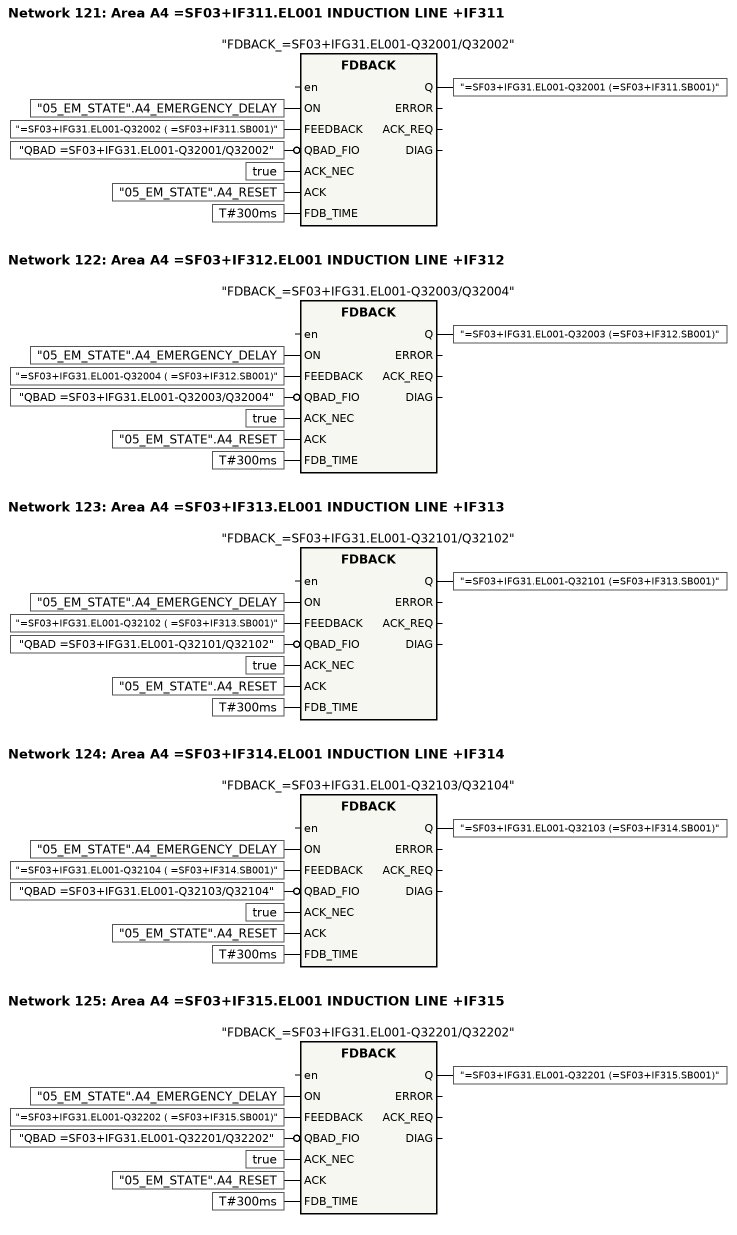
   "FDBACK_=SF03+IFG31.EL001-Q32001/Q32002"(ON := "05_EM_STATE".A4_EMERGENCY_DELAY,   // FDBACK
                           FEEDBACK := "=SF03+IFG31.EL001-Q32002 ( =SF03+IF311.SB001)",
                           QBAD_FIO := NOT "QBAD =SF03+IFG31.EL001-Q32001/Q32002",
                           ACK_NEC := true,
                           ACK := "05_EM_STATE".A4_RESET,
                           FDB_TIME := T#300ms,
                           Q => "=SF03+IFG31.EL001-Q32001 (=SF03+IF311.SB001)");
END_REGION

REGION Network 122: Area A4 =SF03+IF312.EL001 INDUCTION LINE +IF312
   "FDBACK_=SF03+IFG31.EL001-Q32003/Q32004"(ON := "05_EM_STATE".A4_EMERGENCY_DELAY,   // FDBACK
                           FEEDBACK := "=SF03+IFG31.EL001-Q32004 ( =SF03+IF312.SB001)",
                           QBAD_FIO := NOT "QBAD =SF03+IFG31.EL001-Q32003/Q32004",
                           ACK_NEC := true,
                           ACK := "05_EM_STATE".A4_RESET,
                           FDB_TIME := T#300ms,
                           Q => "=SF03+IFG31.EL001-Q32003 (=SF03+IF312.SB001)");
END_REGION

REGION Network 123: Area A4 =SF03+IF313.EL001 INDUCTION LINE +IF313
   "FDBACK_=SF03+IFG31.EL001-Q32101/Q32102"(ON := "05_EM_STATE".A4_EMERGENCY_DELAY,   // FDBACK
                           FEEDBACK := "=SF03+IFG31.EL001-Q32102 ( =SF03+IF313.SB001)",
                           QBAD_FIO := NOT "QBAD =SF03+IFG31.EL001-Q32101/Q32102",
                           ACK_NEC := true,
                           ACK := "05_EM_STATE".A4_RESET,
                           FDB_TIME := T#300ms,
                           Q => "=SF03+IFG31.EL001-Q32101 (=SF03+IF313.SB001)");
END_REGION

REGION Network 124: Area A4 =SF03+IF314.EL001 INDUCTION LINE +IF314
   "FDBACK_=SF03+IFG31.EL001-Q32103/Q32104"(ON := "05_EM_STATE".A4_EMERGENCY_DELAY,   // FDBACK
                           FEEDBACK := "=SF03+IFG31.EL001-Q32104 ( =SF03+IF314.SB001)",
                           QBAD_FIO := NOT "QBAD =SF03+IFG31.EL001-Q32103/Q32104",
                           ACK_NEC := true,
                           ACK := "05_EM_STATE".A4_RESET,
                           FDB_TIME := T#300ms,
                           Q => "=SF03+IFG31.EL001-Q32103 (=SF03+IF314.SB001)");
END_REGION

REGION Network 125: Area A4 =SF03+IF315.EL001 INDUCTION LINE +IF315
   "FDBACK_=SF03+IFG31.EL001-Q32201/Q32202"(ON := "05_EM_STATE".A4_EMERGENCY_DELAY,   // FDBACK
                           FEEDBACK := "=SF03+IFG31.EL001-Q32202 ( =SF03+IF315.SB001)",
                           QBAD_FIO := NOT "QBAD =SF03+IFG31.EL001-Q32201/Q32202",
                           ACK_NEC := true,
                           ACK := "05_EM_STATE".A4_RESET,
                           FDB_TIME := T#300ms,
                           Q => "=SF03+IFG31.EL001-Q32201 (=SF03+IF315.SB001)");
END_REGION

REGION Network 126: Area A4 =SF04+IF411.EL001 INDUCTION LINE +IF411
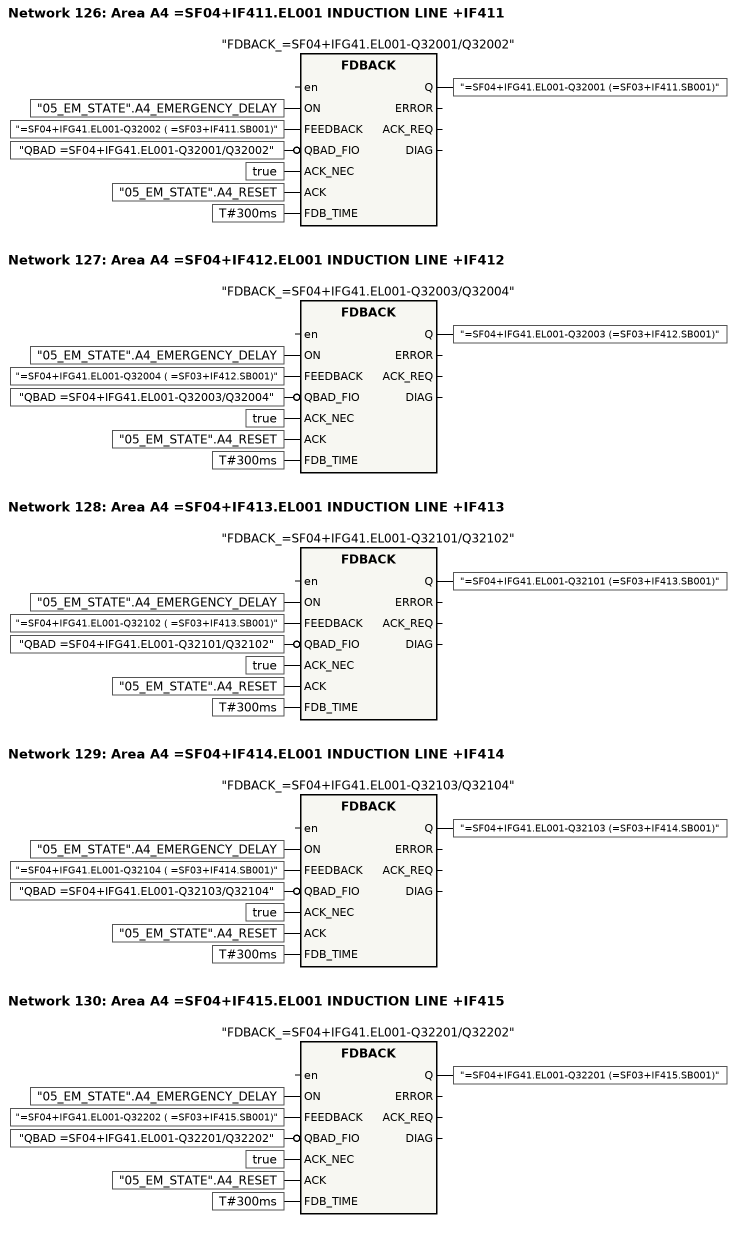
   "FDBACK_=SF04+IFG41.EL001-Q32001/Q32002"(ON := "05_EM_STATE".A4_EMERGENCY_DELAY,   // FDBACK
                           FEEDBACK := "=SF04+IFG41.EL001-Q32002 ( =SF03+IF411.SB001)",
                           QBAD_FIO := NOT "QBAD =SF04+IFG41.EL001-Q32001/Q32002",
                           ACK_NEC := true,
                           ACK := "05_EM_STATE".A4_RESET,
                           FDB_TIME := T#300ms,
                           Q => "=SF04+IFG41.EL001-Q32001 (=SF03+IF411.SB001)");
END_REGION

REGION Network 127: Area A4 =SF04+IF412.EL001 INDUCTION LINE +IF412
   "FDBACK_=SF04+IFG41.EL001-Q32003/Q32004"(ON := "05_EM_STATE".A4_EMERGENCY_DELAY,   // FDBACK
                           FEEDBACK := "=SF04+IFG41.EL001-Q32004 ( =SF03+IF412.SB001)",
                           QBAD_FIO := NOT "QBAD =SF04+IFG41.EL001-Q32003/Q32004",
                           ACK_NEC := true,
                           ACK := "05_EM_STATE".A4_RESET,
                           FDB_TIME := T#300ms,
                           Q => "=SF04+IFG41.EL001-Q32003 (=SF03+IF412.SB001)");
END_REGION

REGION Network 128: Area A4 =SF04+IF413.EL001 INDUCTION LINE +IF413
   "FDBACK_=SF04+IFG41.EL001-Q32101/Q32102"(ON := "05_EM_STATE".A4_EMERGENCY_DELAY,   // FDBACK
                           FEEDBACK := "=SF04+IFG41.EL001-Q32102 ( =SF03+IF413.SB001)",
                           QBAD_FIO := NOT "QBAD =SF04+IFG41.EL001-Q32101/Q32102",
                           ACK_NEC := true,
                           ACK := "05_EM_STATE".A4_RESET,
                           FDB_TIME := T#300ms,
                           Q => "=SF04+IFG41.EL001-Q32101 (=SF03+IF413.SB001)");
END_REGION

REGION Network 129: Area A4 =SF04+IF414.EL001 INDUCTION LINE +IF414
   "FDBACK_=SF04+IFG41.EL001-Q32103/Q32104"(ON := "05_EM_STATE".A4_EMERGENCY_DELAY,   // FDBACK
                           FEEDBACK := "=SF04+IFG41.EL001-Q32104 ( =SF03+IF414.SB001)",
                           QBAD_FIO := NOT "QBAD =SF04+IFG41.EL001-Q32103/Q32104",
                           ACK_NEC := true,
                           ACK := "05_EM_STATE".A4_RESET,
                           FDB_TIME := T#300ms,
                           Q => "=SF04+IFG41.EL001-Q32103 (=SF03+IF414.SB001)");
END_REGION

REGION Network 130: Area A4 =SF04+IF415.EL001 INDUCTION LINE +IF415
   "FDBACK_=SF04+IFG41.EL001-Q32201/Q32202"(ON := "05_EM_STATE".A4_EMERGENCY_DELAY,   // FDBACK
                           FEEDBACK := "=SF04+IFG41.EL001-Q32202 ( =SF03+IF415.SB001)",
                           QBAD_FIO := NOT "QBAD =SF04+IFG41.EL001-Q32201/Q32202",
                           ACK_NEC := true,
                           ACK := "05_EM_STATE".A4_RESET,
                           FDB_TIME := T#300ms,
                           Q => "=SF04+IFG41.EL001-Q32201 (=SF03+IF415.SB001)");
END_REGION

REGION Network 131: Area A4 =SF00+FC011.SB001 ROLLER CONVEYOR CHUTES +FH901/FH902
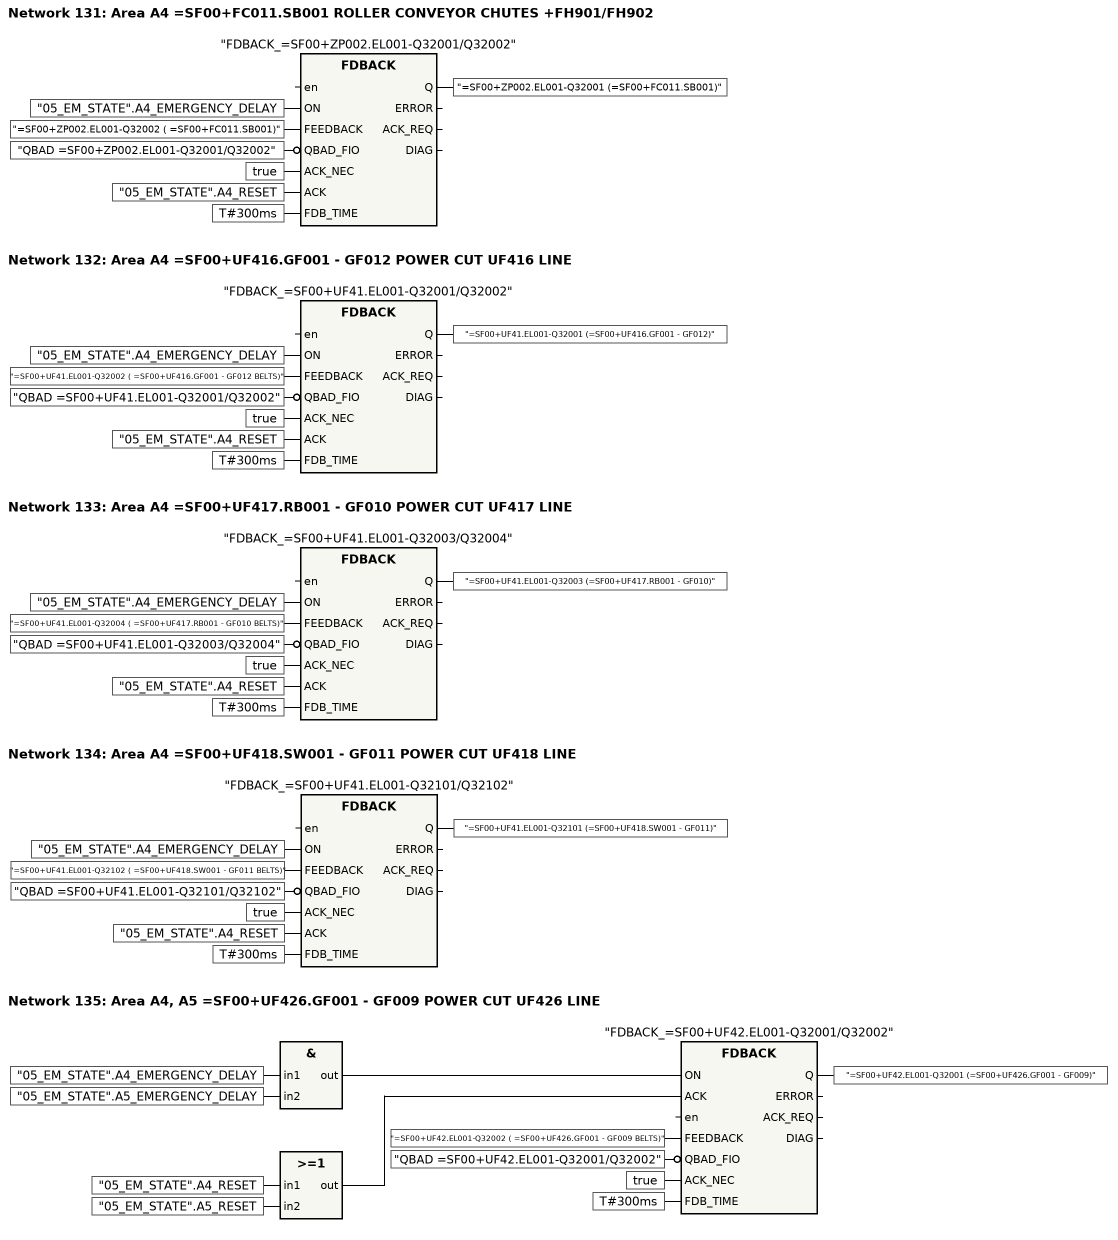
   "FDBACK_=SF00+ZP002.EL001-Q32001/Q32002"(ON := "05_EM_STATE".A4_EMERGENCY_DELAY,   // FDBACK
                           FEEDBACK := "=SF00+ZP002.EL001-Q32002 ( =SF00+FC011.SB001)",
                           QBAD_FIO := NOT "QBAD =SF00+ZP002.EL001-Q32001/Q32002",
                           ACK_NEC := true,
                           ACK := "05_EM_STATE".A4_RESET,
                           FDB_TIME := T#300ms,
                           Q => "=SF00+ZP002.EL001-Q32001 (=SF00+FC011.SB001)");
END_REGION

REGION Network 132: Area A4 =SF00+UF416.GF001 - GF012 POWER CUT UF416 LINE
   "FDBACK_=SF00+UF41.EL001-Q32001/Q32002"(ON := "05_EM_STATE".A4_EMERGENCY_DELAY,   // FDBACK
                           FEEDBACK := "=SF00+UF41.EL001-Q32002 ( =SF00+UF416.GF001 - GF012 BELTS)",
                           QBAD_FIO := NOT "QBAD =SF00+UF41.EL001-Q32001/Q32002",
                           ACK_NEC := true,
                           ACK := "05_EM_STATE".A4_RESET,
                           FDB_TIME := T#300ms,
                           Q => "=SF00+UF41.EL001-Q32001 (=SF00+UF416.GF001 - GF012)");
END_REGION

REGION Network 133: Area A4 =SF00+UF417.RB001 - GF010 POWER CUT UF417 LINE
   "FDBACK_=SF00+UF41.EL001-Q32003/Q32004"(ON := "05_EM_STATE".A4_EMERGENCY_DELAY,   // FDBACK
                           FEEDBACK := "=SF00+UF41.EL001-Q32004 ( =SF00+UF417.RB001 - GF010 BELTS)",
                           QBAD_FIO := NOT "QBAD =SF00+UF41.EL001-Q32003/Q32004",
                           ACK_NEC := true,
                           ACK := "05_EM_STATE".A4_RESET,
                           FDB_TIME := T#300ms,
                           Q => "=SF00+UF41.EL001-Q32003 (=SF00+UF417.RB001 - GF010)");
END_REGION

REGION Network 134: Area A4 =SF00+UF418.SW001 - GF011 POWER CUT UF418 LINE
   "FDBACK_=SF00+UF41.EL001-Q32101/Q32102"(ON := "05_EM_STATE".A4_EMERGENCY_DELAY,   // FDBACK
                           FEEDBACK := "=SF00+UF41.EL001-Q32102 ( =SF00+UF418.SW001 - GF011 BELTS)",
                           QBAD_FIO := NOT "QBAD =SF00+UF41.EL001-Q32101/Q32102",
                           ACK_NEC := true,
                           ACK := "05_EM_STATE".A4_RESET,
                           FDB_TIME := T#300ms,
                           Q => "=SF00+UF41.EL001-Q32101 (=SF00+UF418.SW001 - GF011)");
END_REGION

REGION Network 135: Area A4, A5 =SF00+UF426.GF001 - GF009 POWER CUT UF426 LINE
   "FDBACK_=SF00+UF42.EL001-Q32001/Q32002"(ON := "05_EM_STATE".A4_EMERGENCY_DELAY AND "05_EM_STATE".A5_EMERGENCY_DELAY,   // FDBACK
                           ACK := "05_EM_STATE".A4_RESET OR "05_EM_STATE".A5_RESET,
                           FEEDBACK := "=SF00+UF42.EL001-Q32002 ( =SF00+UF426.GF001 - GF009 BELTS)",
                           QBAD_FIO := NOT "QBAD =SF00+UF42.EL001-Q32001/Q32002",
                           ACK_NEC := true,
                           FDB_TIME := T#300ms,
                           Q => "=SF00+UF42.EL001-Q32001 (=SF00+UF426.GF001 - GF009)");
END_REGION

REGION Network 136: Area A4 =SF00+UF428.RB001 - GF010 POWER CUT UF428 LINE
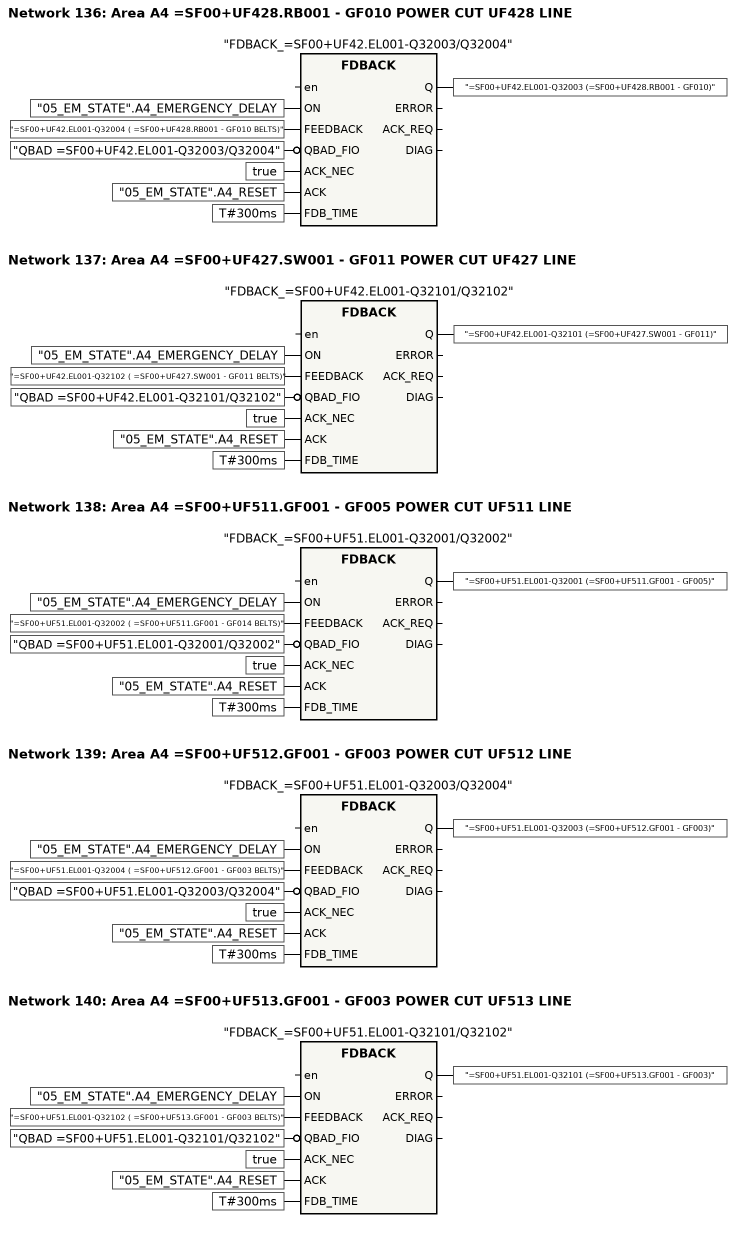
   "FDBACK_=SF00+UF42.EL001-Q32003/Q32004"(ON := "05_EM_STATE".A4_EMERGENCY_DELAY,   // FDBACK
                           FEEDBACK := "=SF00+UF42.EL001-Q32004 ( =SF00+UF428.RB001 - GF010 BELTS)",
                           QBAD_FIO := NOT "QBAD =SF00+UF42.EL001-Q32003/Q32004",
                           ACK_NEC := true,
                           ACK := "05_EM_STATE".A4_RESET,
                           FDB_TIME := T#300ms,
                           Q => "=SF00+UF42.EL001-Q32003 (=SF00+UF428.RB001 - GF010)");
END_REGION

REGION Network 137: Area A4 =SF00+UF427.SW001 - GF011 POWER CUT UF427 LINE
   "FDBACK_=SF00+UF42.EL001-Q32101/Q32102"(ON := "05_EM_STATE".A4_EMERGENCY_DELAY,   // FDBACK
                           FEEDBACK := "=SF00+UF42.EL001-Q32102 ( =SF00+UF427.SW001 - GF011 BELTS)",
                           QBAD_FIO := NOT "QBAD =SF00+UF42.EL001-Q32101/Q32102",
                           ACK_NEC := true,
                           ACK := "05_EM_STATE".A4_RESET,
                           FDB_TIME := T#300ms,
                           Q => "=SF00+UF42.EL001-Q32101 (=SF00+UF427.SW001 - GF011)");
END_REGION

REGION Network 138: Area A4 =SF00+UF511.GF001 - GF005 POWER CUT UF511 LINE
   "FDBACK_=SF00+UF51.EL001-Q32001/Q32002"(ON := "05_EM_STATE".A4_EMERGENCY_DELAY,   // FDBACK
                           FEEDBACK := "=SF00+UF51.EL001-Q32002 ( =SF00+UF511.GF001 - GF014 BELTS)",
                           QBAD_FIO := NOT "QBAD =SF00+UF51.EL001-Q32001/Q32002",
                           ACK_NEC := true,
                           ACK := "05_EM_STATE".A4_RESET,
                           FDB_TIME := T#300ms,
                           Q => "=SF00+UF51.EL001-Q32001 (=SF00+UF511.GF001 - GF005)");
END_REGION

REGION Network 139: Area A4 =SF00+UF512.GF001 - GF003 POWER CUT UF512 LINE
   "FDBACK_=SF00+UF51.EL001-Q32003/Q32004"(ON := "05_EM_STATE".A4_EMERGENCY_DELAY,   // FDBACK
                           FEEDBACK := "=SF00+UF51.EL001-Q32004 ( =SF00+UF512.GF001 - GF003 BELTS)",
                           QBAD_FIO := NOT "QBAD =SF00+UF51.EL001-Q32003/Q32004",
                           ACK_NEC := true,
                           ACK := "05_EM_STATE".A4_RESET,
                           FDB_TIME := T#300ms,
                           Q => "=SF00+UF51.EL001-Q32003 (=SF00+UF512.GF001 - GF003)");
END_REGION

REGION Network 140: Area A4 =SF00+UF513.GF001 - GF003 POWER CUT UF513 LINE
   "FDBACK_=SF00+UF51.EL001-Q32101/Q32102"(ON := "05_EM_STATE".A4_EMERGENCY_DELAY,   // FDBACK
                           FEEDBACK := "=SF00+UF51.EL001-Q32102 ( =SF00+UF513.GF001 - GF003 BELTS)",
                           QBAD_FIO := NOT "QBAD =SF00+UF51.EL001-Q32101/Q32102",
                           ACK_NEC := true,
                           ACK := "05_EM_STATE".A4_RESET,
                           FDB_TIME := T#300ms,
                           Q => "=SF00+UF51.EL001-Q32101 (=SF00+UF513.GF001 - GF003)");
END_REGION

REGION Network 141: Area A4, L15 =SF00+UF511.VS015 POWER CUT UF511 VERTICAL SWITCH
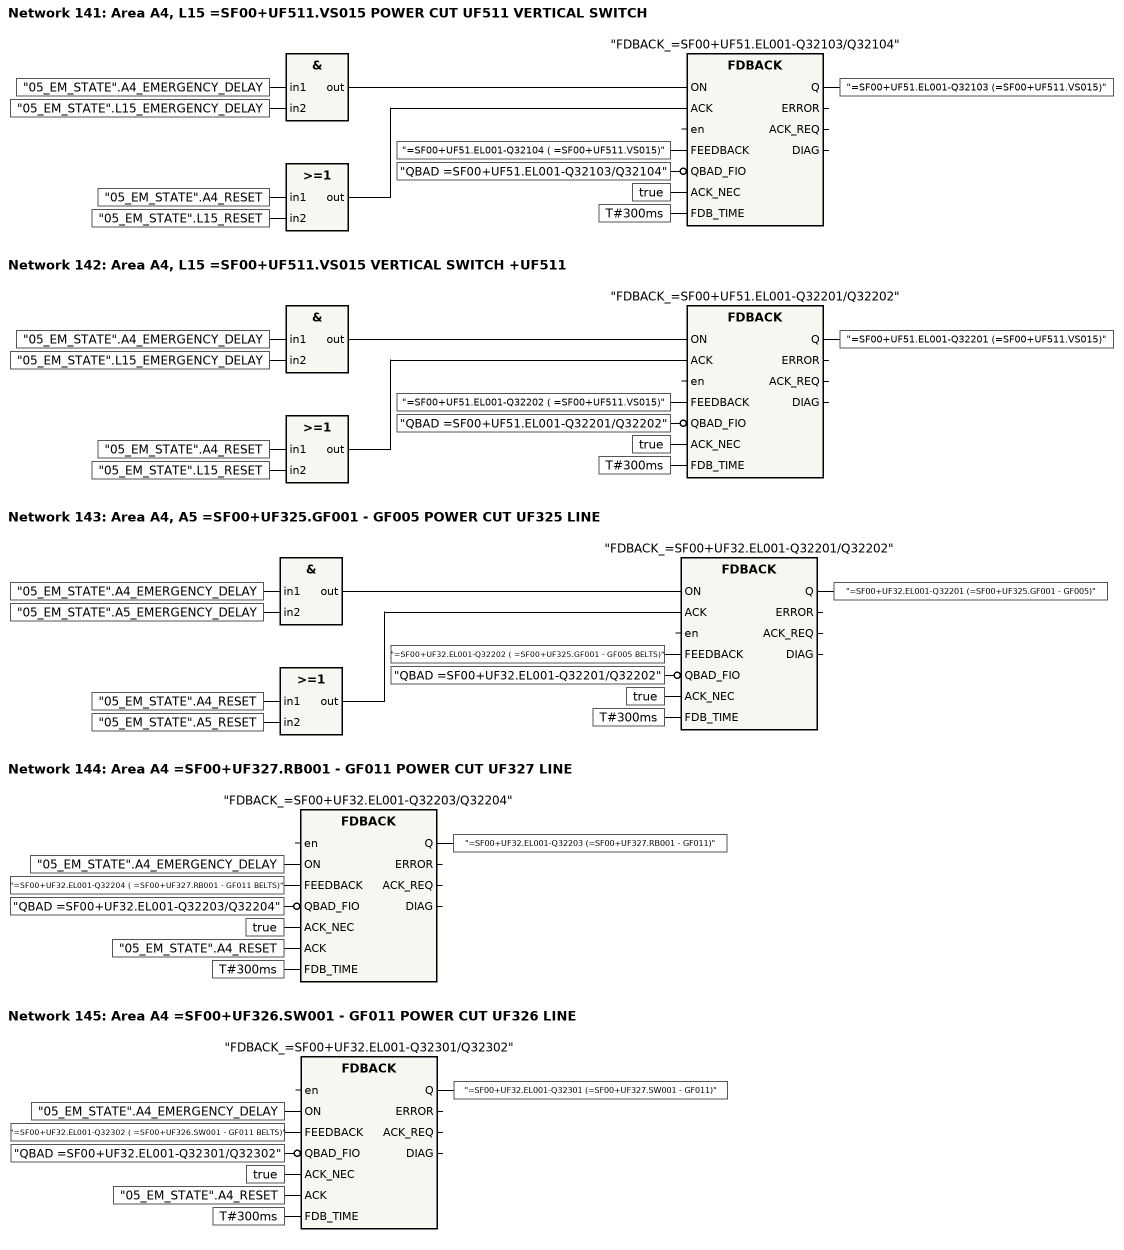
   "FDBACK_=SF00+UF51.EL001-Q32103/Q32104"(ON := "05_EM_STATE".A4_EMERGENCY_DELAY AND "05_EM_STATE".L15_EMERGENCY_DELAY,   // FDBACK
                           ACK := "05_EM_STATE".A4_RESET OR "05_EM_STATE".L15_RESET,
                           FEEDBACK := "=SF00+UF51.EL001-Q32104 ( =SF00+UF511.VS015)",
                           QBAD_FIO := NOT "QBAD =SF00+UF51.EL001-Q32103/Q32104",
                           ACK_NEC := true,
                           FDB_TIME := T#300ms,
                           Q => "=SF00+UF51.EL001-Q32103 (=SF00+UF511.VS015)");
END_REGION

REGION Network 142: Area A4, L15 =SF00+UF511.VS015 VERTICAL SWITCH +UF511
   "FDBACK_=SF00+UF51.EL001-Q32201/Q32202"(ON := "05_EM_STATE".A4_EMERGENCY_DELAY AND "05_EM_STATE".L15_EMERGENCY_DELAY,   // FDBACK
                           ACK := "05_EM_STATE".A4_RESET OR "05_EM_STATE".L15_RESET,
                           FEEDBACK := "=SF00+UF51.EL001-Q32202 ( =SF00+UF511.VS015)",
                           QBAD_FIO := NOT "QBAD =SF00+UF51.EL001-Q32201/Q32202",
                           ACK_NEC := true,
                           FDB_TIME := T#300ms,
                           Q => "=SF00+UF51.EL001-Q32201 (=SF00+UF511.VS015)");
END_REGION

REGION Network 143: Area A4, A5 =SF00+UF325.GF001 - GF005 POWER CUT UF325 LINE
   "FDBACK_=SF00+UF32.EL001-Q32201/Q32202"(ON := "05_EM_STATE".A4_EMERGENCY_DELAY AND "05_EM_STATE".A5_EMERGENCY_DELAY,   // FDBACK
                           ACK := "05_EM_STATE".A4_RESET OR "05_EM_STATE".A5_RESET,
                           FEEDBACK := "=SF00+UF32.EL001-Q32202 ( =SF00+UF325.GF001 - GF005 BELTS)",
                           QBAD_FIO := NOT "QBAD =SF00+UF32.EL001-Q32201/Q32202",
                           ACK_NEC := true,
                           FDB_TIME := T#300ms,
                           Q => "=SF00+UF32.EL001-Q32201 (=SF00+UF325.GF001 - GF005)");
END_REGION

REGION Network 144: Area A4 =SF00+UF327.RB001 - GF011 POWER CUT UF327 LINE
   "FDBACK_=SF00+UF32.EL001-Q32203/Q32204"(ON := "05_EM_STATE".A4_EMERGENCY_DELAY,   // FDBACK
                           FEEDBACK := "=SF00+UF32.EL001-Q32204 ( =SF00+UF327.RB001 - GF011 BELTS)",
                           QBAD_FIO := NOT "QBAD =SF00+UF32.EL001-Q32203/Q32204",
                           ACK_NEC := true,
                           ACK := "05_EM_STATE".A4_RESET,
                           FDB_TIME := T#300ms,
                           Q => "=SF00+UF32.EL001-Q32203 (=SF00+UF327.RB001 - GF011)");
END_REGION

REGION Network 145: Area A4 =SF00+UF326.SW001 - GF011 POWER CUT UF326 LINE
   "FDBACK_=SF00+UF32.EL001-Q32301/Q32302"(ON := "05_EM_STATE".A4_EMERGENCY_DELAY,   // FDBACK
                           FEEDBACK := "=SF00+UF32.EL001-Q32302 ( =SF00+UF326.SW001 - GF011 BELTS)",
                           QBAD_FIO := NOT "QBAD =SF00+UF32.EL001-Q32301/Q32302",
                           ACK_NEC := true,
                           ACK := "05_EM_STATE".A4_RESET,
                           FDB_TIME := T#300ms,
                           Q => "=SF00+UF32.EL001-Q32301 (=SF00+UF327.SW001 - GF011)");
END_REGION

REGION Network 146: Area A4 =SF00+UF317.GF001 - GF012 POWER CUT UF317 LINE
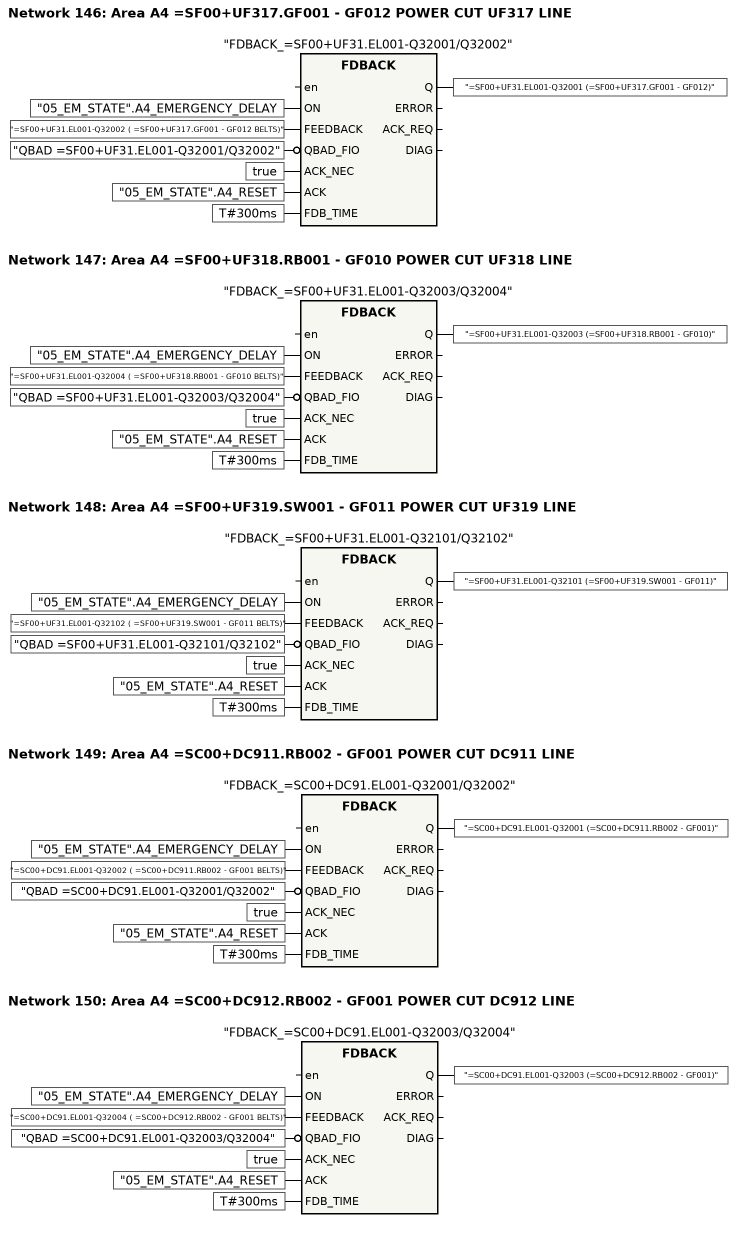
   "FDBACK_=SF00+UF31.EL001-Q32001/Q32002"(ON := "05_EM_STATE".A4_EMERGENCY_DELAY,   // FDBACK
                           FEEDBACK := "=SF00+UF31.EL001-Q32002 ( =SF00+UF317.GF001 - GF012 BELTS)",
                           QBAD_FIO := NOT "QBAD =SF00+UF31.EL001-Q32001/Q32002",
                           ACK_NEC := true,
                           ACK := "05_EM_STATE".A4_RESET,
                           FDB_TIME := T#300ms,
                           Q => "=SF00+UF31.EL001-Q32001 (=SF00+UF317.GF001 - GF012)");
END_REGION

REGION Network 147: Area A4 =SF00+UF318.RB001 - GF010 POWER CUT UF318 LINE
   "FDBACK_=SF00+UF31.EL001-Q32003/Q32004"(ON := "05_EM_STATE".A4_EMERGENCY_DELAY,   // FDBACK
                           FEEDBACK := "=SF00+UF31.EL001-Q32004 ( =SF00+UF318.RB001 - GF010 BELTS)",
                           QBAD_FIO := NOT "QBAD =SF00+UF31.EL001-Q32003/Q32004",
                           ACK_NEC := true,
                           ACK := "05_EM_STATE".A4_RESET,
                           FDB_TIME := T#300ms,
                           Q => "=SF00+UF31.EL001-Q32003 (=SF00+UF318.RB001 - GF010)");
END_REGION

REGION Network 148: Area A4 =SF00+UF319.SW001 - GF011 POWER CUT UF319 LINE
   "FDBACK_=SF00+UF31.EL001-Q32101/Q32102"(ON := "05_EM_STATE".A4_EMERGENCY_DELAY,   // FDBACK
                           FEEDBACK := "=SF00+UF31.EL001-Q32102 ( =SF00+UF319.SW001 - GF011 BELTS)",
                           QBAD_FIO := NOT "QBAD =SF00+UF31.EL001-Q32101/Q32102",
                           ACK_NEC := true,
                           ACK := "05_EM_STATE".A4_RESET,
                           FDB_TIME := T#300ms,
                           Q => "=SF00+UF31.EL001-Q32101 (=SF00+UF319.SW001 - GF011)");
END_REGION

REGION Network 149: Area A4 =SC00+DC911.RB002 - GF001 POWER CUT DC911 LINE
   "FDBACK_=SC00+DC91.EL001-Q32001/Q32002"(ON := "05_EM_STATE".A4_EMERGENCY_DELAY,   // FDBACK
                           FEEDBACK := "=SC00+DC91.EL001-Q32002 ( =SC00+DC911.RB002 - GF001 BELTS)",
                           QBAD_FIO := NOT "QBAD =SC00+DC91.EL001-Q32001/Q32002",
                           ACK_NEC := true,
                           ACK := "05_EM_STATE".A4_RESET,
                           FDB_TIME := T#300ms,
                           Q => "=SC00+DC91.EL001-Q32001 (=SC00+DC911.RB002 - GF001)");
END_REGION

REGION Network 150: Area A4 =SC00+DC912.RB002 - GF001 POWER CUT DC912 LINE
   "FDBACK_=SC00+DC91.EL001-Q32003/Q32004"(ON := "05_EM_STATE".A4_EMERGENCY_DELAY,   // FDBACK
                           FEEDBACK := "=SC00+DC91.EL001-Q32004 ( =SC00+DC912.RB002 - GF001 BELTS)",
                           QBAD_FIO := NOT "QBAD =SC00+DC91.EL001-Q32003/Q32004",
                           ACK_NEC := true,
                           ACK := "05_EM_STATE".A4_RESET,
                           FDB_TIME := T#300ms,
                           Q => "=SC00+DC91.EL001-Q32003 (=SC00+DC912.RB002 - GF001)");
END_REGION

REGION Network 151: Area A4 =SC00+DC913.RB002 - GF001 POWER CUT DC913 LINE
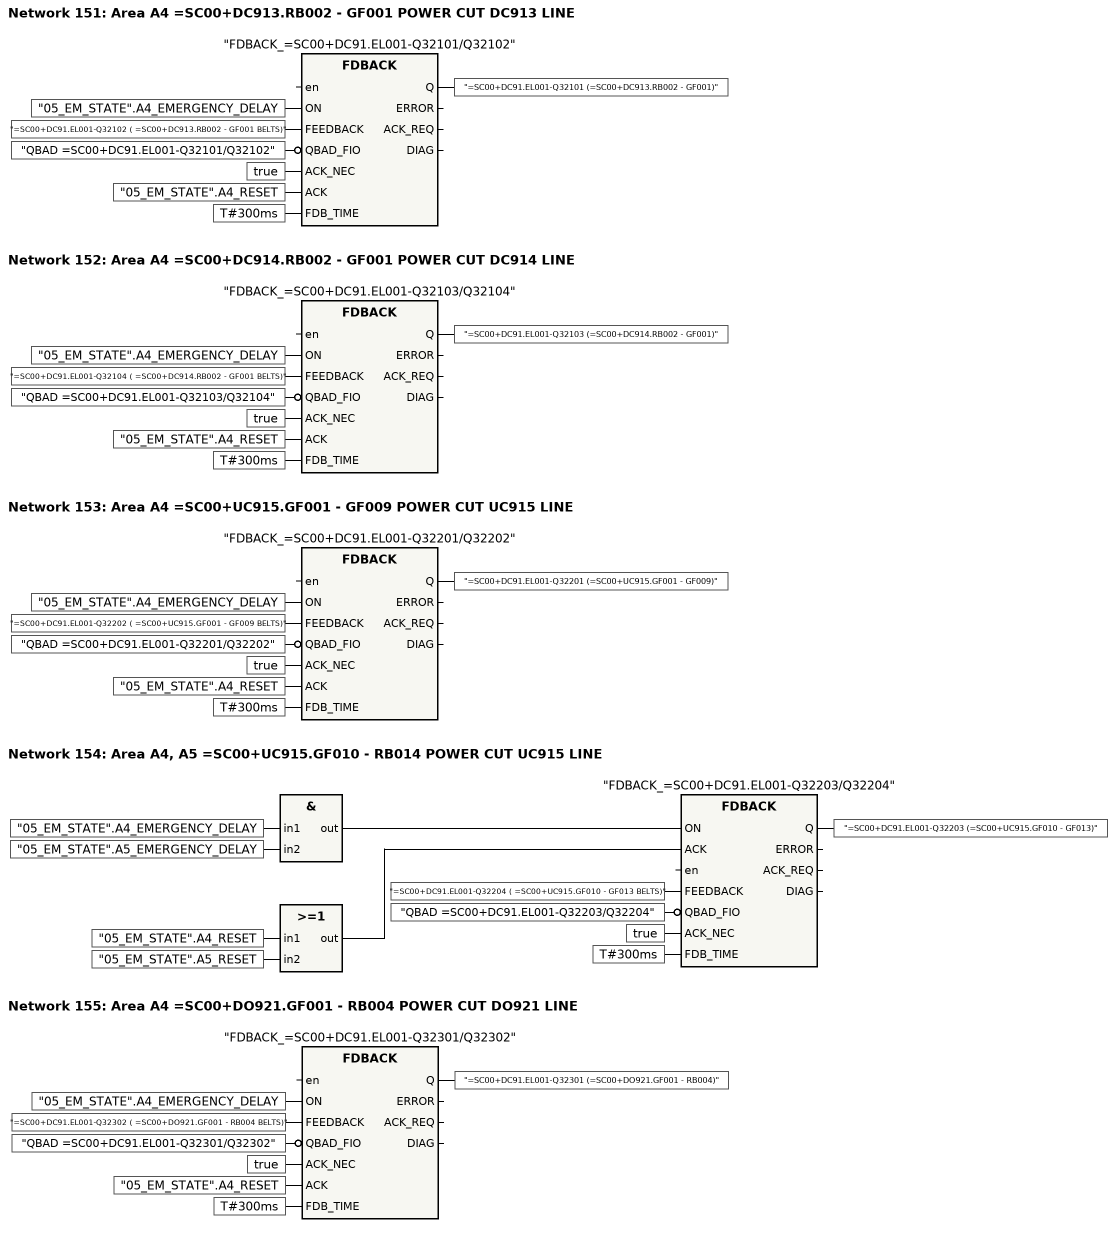
   "FDBACK_=SC00+DC91.EL001-Q32101/Q32102"(ON := "05_EM_STATE".A4_EMERGENCY_DELAY,   // FDBACK
                           FEEDBACK := "=SC00+DC91.EL001-Q32102 ( =SC00+DC913.RB002 - GF001 BELTS)",
                           QBAD_FIO := NOT "QBAD =SC00+DC91.EL001-Q32101/Q32102",
                           ACK_NEC := true,
                           ACK := "05_EM_STATE".A4_RESET,
                           FDB_TIME := T#300ms,
                           Q => "=SC00+DC91.EL001-Q32101 (=SC00+DC913.RB002 - GF001)");
END_REGION

REGION Network 152: Area A4 =SC00+DC914.RB002 - GF001 POWER CUT DC914 LINE
   "FDBACK_=SC00+DC91.EL001-Q32103/Q32104"(ON := "05_EM_STATE".A4_EMERGENCY_DELAY,   // FDBACK
                           FEEDBACK := "=SC00+DC91.EL001-Q32104 ( =SC00+DC914.RB002 - GF001 BELTS)",
                           QBAD_FIO := NOT "QBAD =SC00+DC91.EL001-Q32103/Q32104",
                           ACK_NEC := true,
                           ACK := "05_EM_STATE".A4_RESET,
                           FDB_TIME := T#300ms,
                           Q => "=SC00+DC91.EL001-Q32103 (=SC00+DC914.RB002 - GF001)");
END_REGION

REGION Network 153: Area A4 =SC00+UC915.GF001 - GF009 POWER CUT UC915 LINE
   "FDBACK_=SC00+DC91.EL001-Q32201/Q32202"(ON := "05_EM_STATE".A4_EMERGENCY_DELAY,   // FDBACK
                           FEEDBACK := "=SC00+DC91.EL001-Q32202 ( =SC00+UC915.GF001 - GF009 BELTS)",
                           QBAD_FIO := NOT "QBAD =SC00+DC91.EL001-Q32201/Q32202",
                           ACK_NEC := true,
                           ACK := "05_EM_STATE".A4_RESET,
                           FDB_TIME := T#300ms,
                           Q => "=SC00+DC91.EL001-Q32201 (=SC00+UC915.GF001 - GF009)");
END_REGION

REGION Network 154: Area A4, A5 =SC00+UC915.GF010 - RB014 POWER CUT UC915 LINE
   "FDBACK_=SC00+DC91.EL001-Q32203/Q32204"(ON := "05_EM_STATE".A4_EMERGENCY_DELAY AND "05_EM_STATE".A5_EMERGENCY_DELAY,   // FDBACK
                           ACK := "05_EM_STATE".A4_RESET OR "05_EM_STATE".A5_RESET,
                           FEEDBACK := "=SC00+DC91.EL001-Q32204 ( =SC00+UC915.GF010 - GF013 BELTS)",
                           QBAD_FIO := NOT "QBAD =SC00+DC91.EL001-Q32203/Q32204",
                           ACK_NEC := true,
                           FDB_TIME := T#300ms,
                           Q => "=SC00+DC91.EL001-Q32203 (=SC00+UC915.GF010 - GF013)");
END_REGION

REGION Network 155: Area A4 =SC00+DO921.GF001 - RB004 POWER CUT DO921 LINE
   "FDBACK_=SC00+DC91.EL001-Q32301/Q32302"(ON := "05_EM_STATE".A4_EMERGENCY_DELAY,   // FDBACK
                           FEEDBACK := "=SC00+DC91.EL001-Q32302 ( =SC00+DO921.GF001 - RB004 BELTS)",
                           QBAD_FIO := NOT "QBAD =SC00+DC91.EL001-Q32301/Q32302",
                           ACK_NEC := true,
                           ACK := "05_EM_STATE".A4_RESET,
                           FDB_TIME := T#300ms,
                           Q => "=SC00+DC91.EL001-Q32301 (=SC00+DO921.GF001 - RB004)");
END_REGION

REGION Network 156: Area A4, A5 =SC00+UC291.GF001 - RB010 POWER CUT UC291 LINE
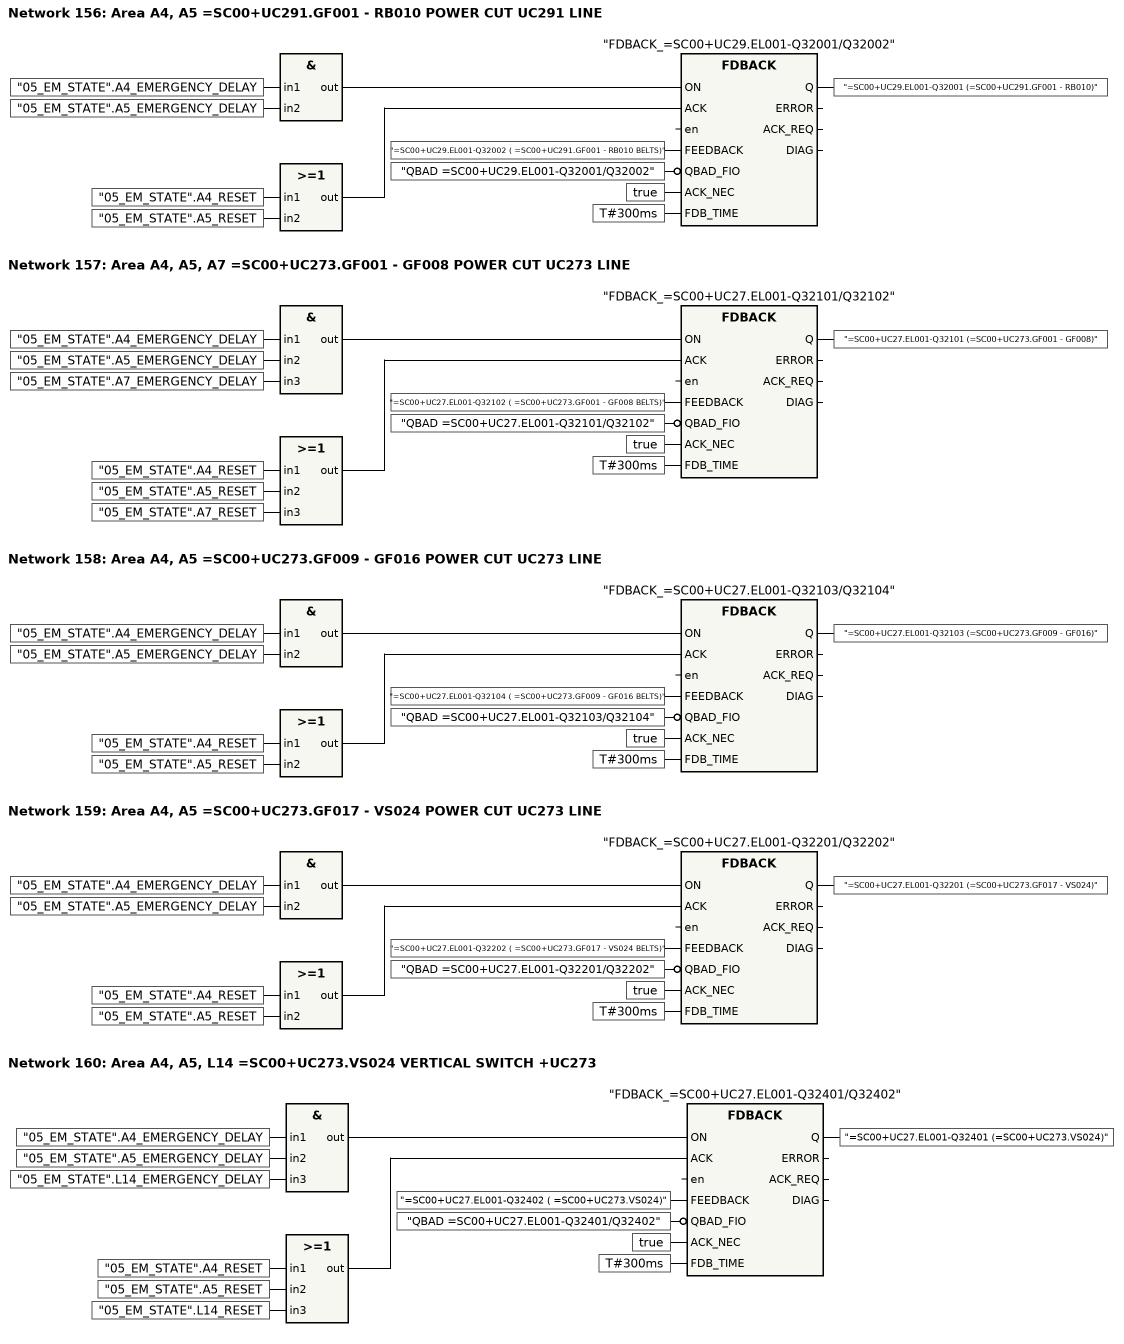
   "FDBACK_=SC00+UC29.EL001-Q32001/Q32002"(ON := "05_EM_STATE".A4_EMERGENCY_DELAY AND "05_EM_STATE".A5_EMERGENCY_DELAY,   // FDBACK
                           ACK := "05_EM_STATE".A4_RESET OR "05_EM_STATE".A5_RESET,
                           FEEDBACK := "=SC00+UC29.EL001-Q32002 ( =SC00+UC291.GF001 - RB010 BELTS)",
                           QBAD_FIO := NOT "QBAD =SC00+UC29.EL001-Q32001/Q32002",
                           ACK_NEC := true,
                           FDB_TIME := T#300ms,
                           Q => "=SC00+UC29.EL001-Q32001 (=SC00+UC291.GF001 - RB010)");
END_REGION

REGION Network 157: Area A4, A5, A7 =SC00+UC273.GF001 - GF008 POWER CUT UC273 LINE
   "FDBACK_=SC00+UC27.EL001-Q32101/Q32102"(ON := "05_EM_STATE".A4_EMERGENCY_DELAY AND "05_EM_STATE".A5_EMERGENCY_DELAY AND "05_EM_STATE".A7_EMERGENCY_DELAY,   // FDBACK
                           ACK := "05_EM_STATE".A4_RESET OR "05_EM_STATE".A5_RESET OR "05_EM_STATE".A7_RESET,
                           FEEDBACK := "=SC00+UC27.EL001-Q32102 ( =SC00+UC273.GF001 - GF008 BELTS)",
                           QBAD_FIO := NOT "QBAD =SC00+UC27.EL001-Q32101/Q32102",
                           ACK_NEC := true,
                           FDB_TIME := T#300ms,
                           Q => "=SC00+UC27.EL001-Q32101 (=SC00+UC273.GF001 - GF008)");
END_REGION

REGION Network 158: Area A4, A5 =SC00+UC273.GF009 - GF016 POWER CUT UC273 LINE
   "FDBACK_=SC00+UC27.EL001-Q32103/Q32104"(ON := "05_EM_STATE".A4_EMERGENCY_DELAY AND "05_EM_STATE".A5_EMERGENCY_DELAY,   // FDBACK
                           ACK := "05_EM_STATE".A4_RESET OR "05_EM_STATE".A5_RESET,
                           FEEDBACK := "=SC00+UC27.EL001-Q32104 ( =SC00+UC273.GF009 - GF016 BELTS)",
                           QBAD_FIO := NOT "QBAD =SC00+UC27.EL001-Q32103/Q32104",
                           ACK_NEC := true,
                           FDB_TIME := T#300ms,
                           Q => "=SC00+UC27.EL001-Q32103 (=SC00+UC273.GF009 - GF016)");
END_REGION

REGION Network 159: Area A4, A5 =SC00+UC273.GF017 - VS024 POWER CUT UC273 LINE
   "FDBACK_=SC00+UC27.EL001-Q32201/Q32202"(ON := "05_EM_STATE".A4_EMERGENCY_DELAY AND "05_EM_STATE".A5_EMERGENCY_DELAY,   // FDBACK
                           ACK := "05_EM_STATE".A4_RESET OR "05_EM_STATE".A5_RESET,
                           FEEDBACK := "=SC00+UC27.EL001-Q32202 ( =SC00+UC273.GF017 - VS024 BELTS)",
                           QBAD_FIO := NOT "QBAD =SC00+UC27.EL001-Q32201/Q32202",
                           ACK_NEC := true,
                           FDB_TIME := T#300ms,
                           Q => "=SC00+UC27.EL001-Q32201 (=SC00+UC273.GF017 - VS024)");
END_REGION

REGION Network 160: Area A4, A5, L14 =SC00+UC273.VS024 VERTICAL SWITCH +UC273
   "FDBACK_=SC00+UC27.EL001-Q32401/Q32402"(ON := "05_EM_STATE".A4_EMERGENCY_DELAY AND "05_EM_STATE".A5_EMERGENCY_DELAY AND "05_EM_STATE".L14_EMERGENCY_DELAY,   // FDBACK
                           ACK := "05_EM_STATE".A4_RESET OR "05_EM_STATE".A5_RESET OR "05_EM_STATE".L14_RESET,
                           FEEDBACK := "=SC00+UC27.EL001-Q32402 ( =SC00+UC273.VS024)",
                           QBAD_FIO := NOT "QBAD =SC00+UC27.EL001-Q32401/Q32402",
                           ACK_NEC := true,
                           FDB_TIME := T#300ms,
                           Q => "=SC00+UC27.EL001-Q32401 (=SC00+UC273.VS024)");
END_REGION

REGION Network 161: Area A4, A5, L14 =SC00+UC273.VS024 VERTICAL SWITCH +UC273
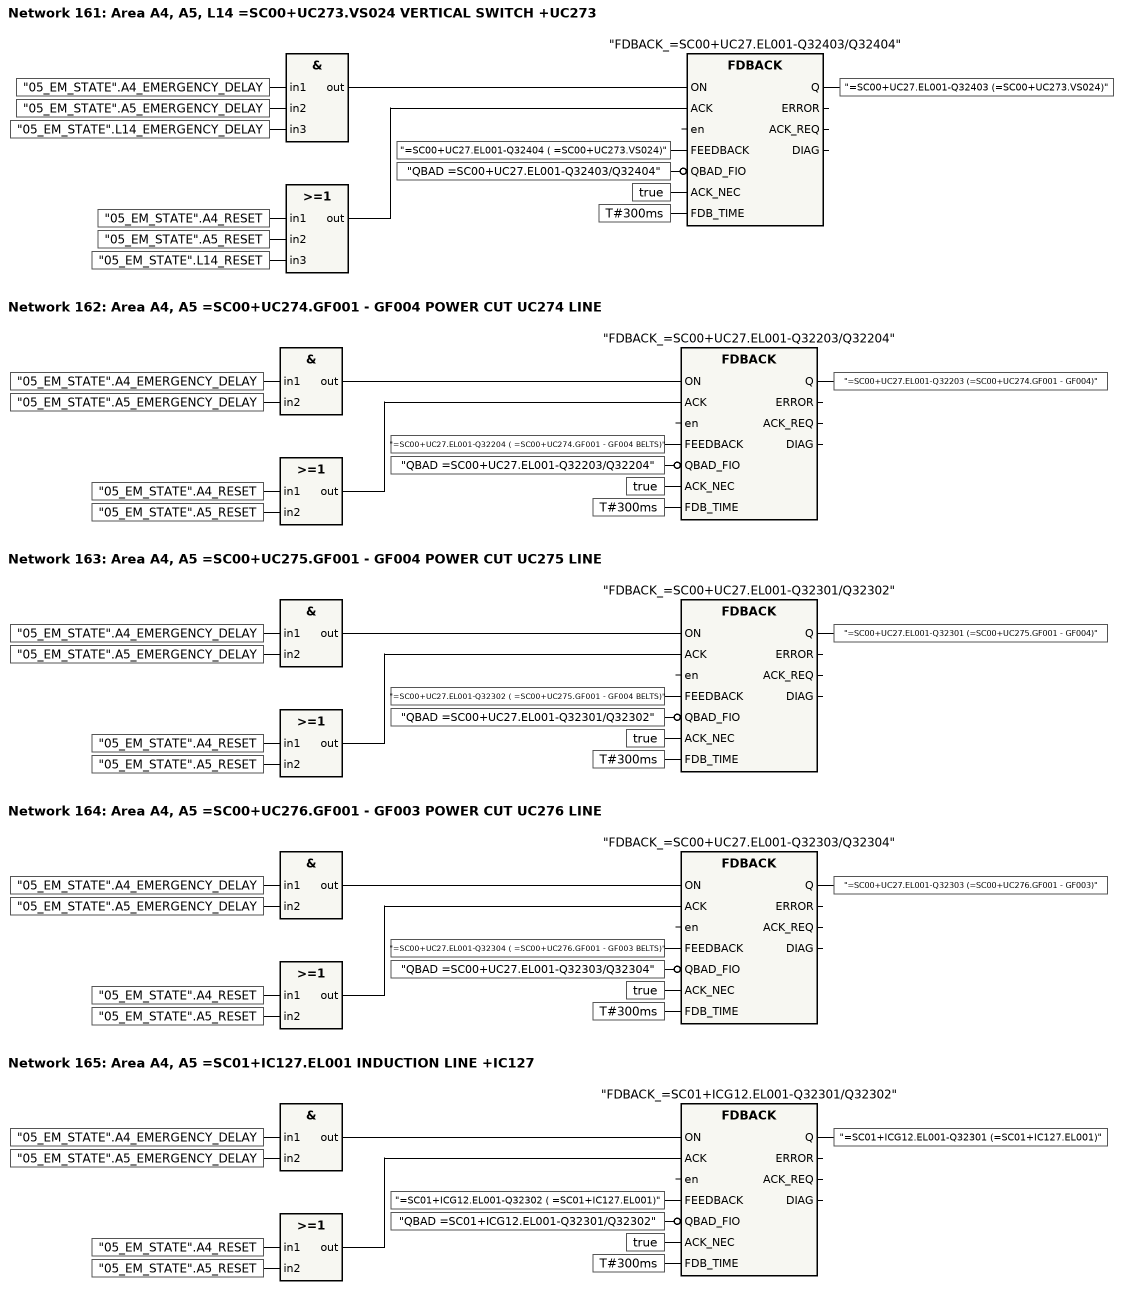
   "FDBACK_=SC00+UC27.EL001-Q32403/Q32404"(ON := "05_EM_STATE".A4_EMERGENCY_DELAY AND "05_EM_STATE".A5_EMERGENCY_DELAY AND "05_EM_STATE".L14_EMERGENCY_DELAY,   // FDBACK
                           ACK := "05_EM_STATE".A4_RESET OR "05_EM_STATE".A5_RESET OR "05_EM_STATE".L14_RESET,
                           FEEDBACK := "=SC00+UC27.EL001-Q32404 ( =SC00+UC273.VS024)",
                           QBAD_FIO := NOT "QBAD =SC00+UC27.EL001-Q32403/Q32404",
                           ACK_NEC := true,
                           FDB_TIME := T#300ms,
                           Q => "=SC00+UC27.EL001-Q32403 (=SC00+UC273.VS024)");
END_REGION

REGION Network 162: Area A4, A5 =SC00+UC274.GF001 - GF004 POWER CUT UC274 LINE
   "FDBACK_=SC00+UC27.EL001-Q32203/Q32204"(ON := "05_EM_STATE".A4_EMERGENCY_DELAY AND "05_EM_STATE".A5_EMERGENCY_DELAY,   // FDBACK
                           ACK := "05_EM_STATE".A4_RESET OR "05_EM_STATE".A5_RESET,
                           FEEDBACK := "=SC00+UC27.EL001-Q32204 ( =SC00+UC274.GF001 - GF004 BELTS)",
                           QBAD_FIO := NOT "QBAD =SC00+UC27.EL001-Q32203/Q32204",
                           ACK_NEC := true,
                           FDB_TIME := T#300ms,
                           Q => "=SC00+UC27.EL001-Q32203 (=SC00+UC274.GF001 - GF004)");
END_REGION

REGION Network 163: Area A4, A5 =SC00+UC275.GF001 - GF004 POWER CUT UC275 LINE
   "FDBACK_=SC00+UC27.EL001-Q32301/Q32302"(ON := "05_EM_STATE".A4_EMERGENCY_DELAY AND "05_EM_STATE".A5_EMERGENCY_DELAY,   // FDBACK
                           ACK := "05_EM_STATE".A4_RESET OR "05_EM_STATE".A5_RESET,
                           FEEDBACK := "=SC00+UC27.EL001-Q32302 ( =SC00+UC275.GF001 - GF004 BELTS)",
                           QBAD_FIO := NOT "QBAD =SC00+UC27.EL001-Q32301/Q32302",
                           ACK_NEC := true,
                           FDB_TIME := T#300ms,
                           Q => "=SC00+UC27.EL001-Q32301 (=SC00+UC275.GF001 - GF004)");
END_REGION

REGION Network 164: Area A4, A5 =SC00+UC276.GF001 - GF003 POWER CUT UC276 LINE
   "FDBACK_=SC00+UC27.EL001-Q32303/Q32304"(ON := "05_EM_STATE".A4_EMERGENCY_DELAY AND "05_EM_STATE".A5_EMERGENCY_DELAY,   // FDBACK
                           ACK := "05_EM_STATE".A4_RESET OR "05_EM_STATE".A5_RESET,
                           FEEDBACK := "=SC00+UC27.EL001-Q32304 ( =SC00+UC276.GF001 - GF003 BELTS)",
                           QBAD_FIO := NOT "QBAD =SC00+UC27.EL001-Q32303/Q32304",
                           ACK_NEC := true,
                           FDB_TIME := T#300ms,
                           Q => "=SC00+UC27.EL001-Q32303 (=SC00+UC276.GF001 - GF003)");
END_REGION

REGION Network 165: Area A4, A5 =SC01+IC127.EL001 INDUCTION LINE +IC127
   "FDBACK_=SC01+ICG12.EL001-Q32301/Q32302"(ON := "05_EM_STATE".A4_EMERGENCY_DELAY AND "05_EM_STATE".A5_EMERGENCY_DELAY,   // FDBACK
                           ACK := "05_EM_STATE".A4_RESET OR "05_EM_STATE".A5_RESET,
                           FEEDBACK := "=SC01+ICG12.EL001-Q32302 ( =SC01+IC127.EL001)",
                           QBAD_FIO := NOT "QBAD =SC01+ICG12.EL001-Q32301/Q32302",
                           ACK_NEC := true,
                           FDB_TIME := T#300ms,
                           Q => "=SC01+ICG12.EL001-Q32301 (=SC01+IC127.EL001)");
END_REGION

REGION Network 166: Area A4, A5 =SC02+IC227.EL001 INDUCTION LINE +IC227
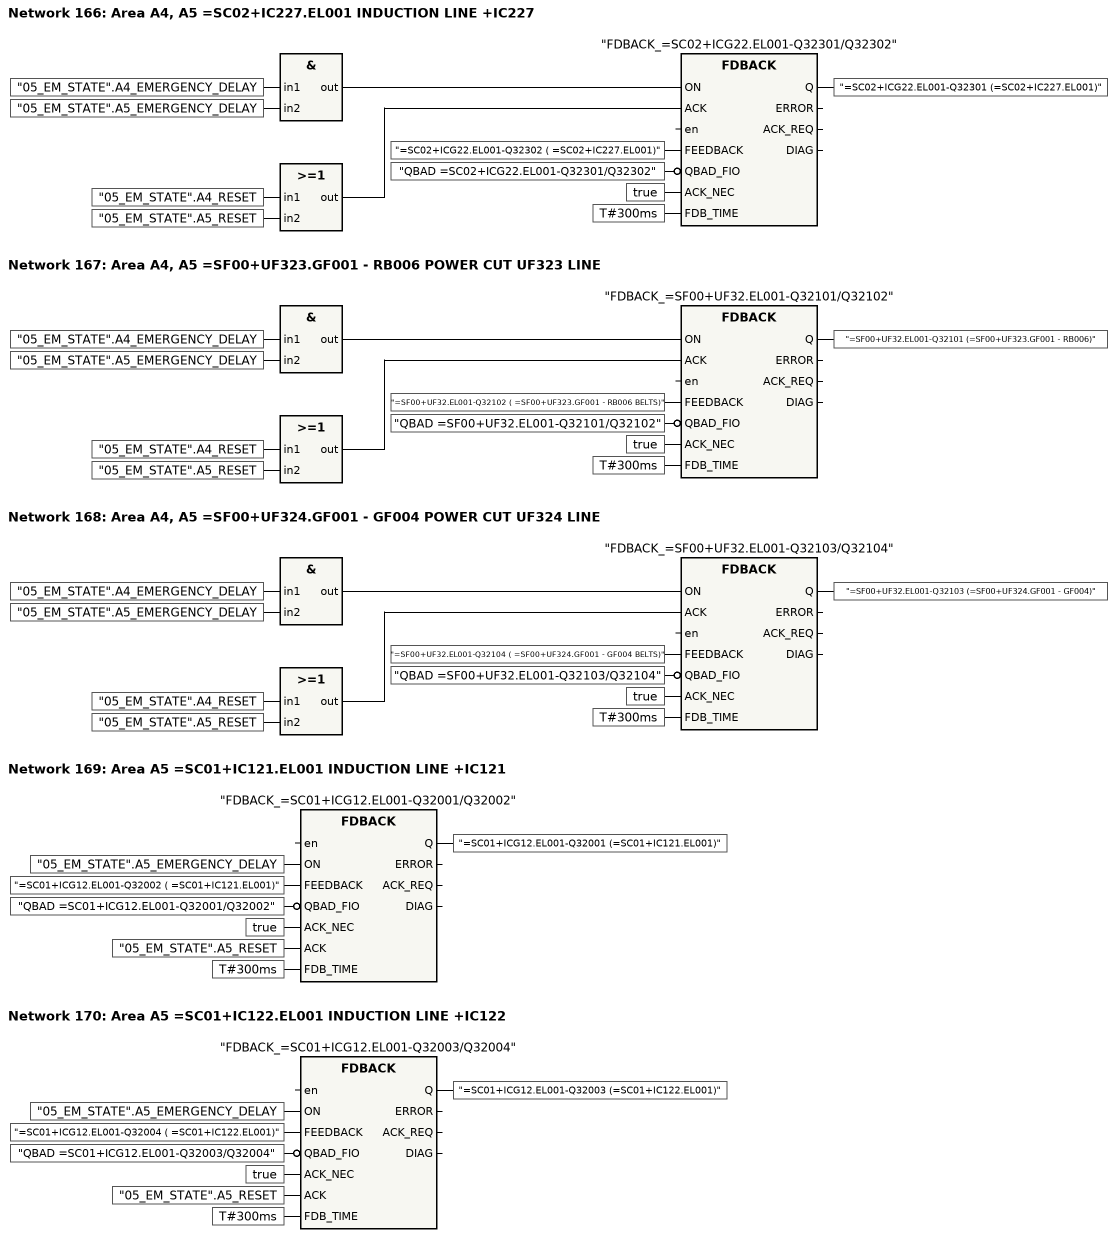
   "FDBACK_=SC02+ICG22.EL001-Q32301/Q32302"(ON := "05_EM_STATE".A4_EMERGENCY_DELAY AND "05_EM_STATE".A5_EMERGENCY_DELAY,   // FDBACK
                           ACK := "05_EM_STATE".A4_RESET OR "05_EM_STATE".A5_RESET,
                           FEEDBACK := "=SC02+ICG22.EL001-Q32302 ( =SC02+IC227.EL001)",
                           QBAD_FIO := NOT "QBAD =SC02+ICG22.EL001-Q32301/Q32302",
                           ACK_NEC := true,
                           FDB_TIME := T#300ms,
                           Q => "=SC02+ICG22.EL001-Q32301 (=SC02+IC227.EL001)");
END_REGION

REGION Network 167: Area A4, A5 =SF00+UF323.GF001 - RB006 POWER CUT UF323 LINE
   "FDBACK_=SF00+UF32.EL001-Q32101/Q32102"(ON := "05_EM_STATE".A4_EMERGENCY_DELAY AND "05_EM_STATE".A5_EMERGENCY_DELAY,   // FDBACK
                           ACK := "05_EM_STATE".A4_RESET OR "05_EM_STATE".A5_RESET,
                           FEEDBACK := "=SF00+UF32.EL001-Q32102 ( =SF00+UF323.GF001 - RB006 BELTS)",
                           QBAD_FIO := NOT "QBAD =SF00+UF32.EL001-Q32101/Q32102",
                           ACK_NEC := true,
                           FDB_TIME := T#300ms,
                           Q => "=SF00+UF32.EL001-Q32101 (=SF00+UF323.GF001 - RB006)");
END_REGION

REGION Network 168: Area A4, A5 =SF00+UF324.GF001 - GF004 POWER CUT UF324 LINE
   "FDBACK_=SF00+UF32.EL001-Q32103/Q32104"(ON := "05_EM_STATE".A4_EMERGENCY_DELAY AND "05_EM_STATE".A5_EMERGENCY_DELAY,   // FDBACK
                           ACK := "05_EM_STATE".A4_RESET OR "05_EM_STATE".A5_RESET,
                           FEEDBACK := "=SF00+UF32.EL001-Q32104 ( =SF00+UF324.GF001 - GF004 BELTS)",
                           QBAD_FIO := NOT "QBAD =SF00+UF32.EL001-Q32103/Q32104",
                           ACK_NEC := true,
                           FDB_TIME := T#300ms,
                           Q => "=SF00+UF32.EL001-Q32103 (=SF00+UF324.GF001 - GF004)");
END_REGION

REGION Network 169: Area A5 =SC01+IC121.EL001 INDUCTION LINE +IC121
   "FDBACK_=SC01+ICG12.EL001-Q32001/Q32002"(ON := "05_EM_STATE".A5_EMERGENCY_DELAY,   // FDBACK
                           FEEDBACK := "=SC01+ICG12.EL001-Q32002 ( =SC01+IC121.EL001)",
                           QBAD_FIO := NOT "QBAD =SC01+ICG12.EL001-Q32001/Q32002",
                           ACK_NEC := true,
                           ACK := "05_EM_STATE".A5_RESET,
                           FDB_TIME := T#300ms,
                           Q => "=SC01+ICG12.EL001-Q32001 (=SC01+IC121.EL001)");
END_REGION

REGION Network 170: Area A5 =SC01+IC122.EL001 INDUCTION LINE +IC122
   "FDBACK_=SC01+ICG12.EL001-Q32003/Q32004"(ON := "05_EM_STATE".A5_EMERGENCY_DELAY,   // FDBACK
                           FEEDBACK := "=SC01+ICG12.EL001-Q32004 ( =SC01+IC122.EL001)",
                           QBAD_FIO := NOT "QBAD =SC01+ICG12.EL001-Q32003/Q32004",
                           ACK_NEC := true,
                           ACK := "05_EM_STATE".A5_RESET,
                           FDB_TIME := T#300ms,
                           Q => "=SC01+ICG12.EL001-Q32003 (=SC01+IC122.EL001)");
END_REGION

REGION Network 171: Area A5 =SC01+IC123.EL001 INDUCTION LINE +IC123
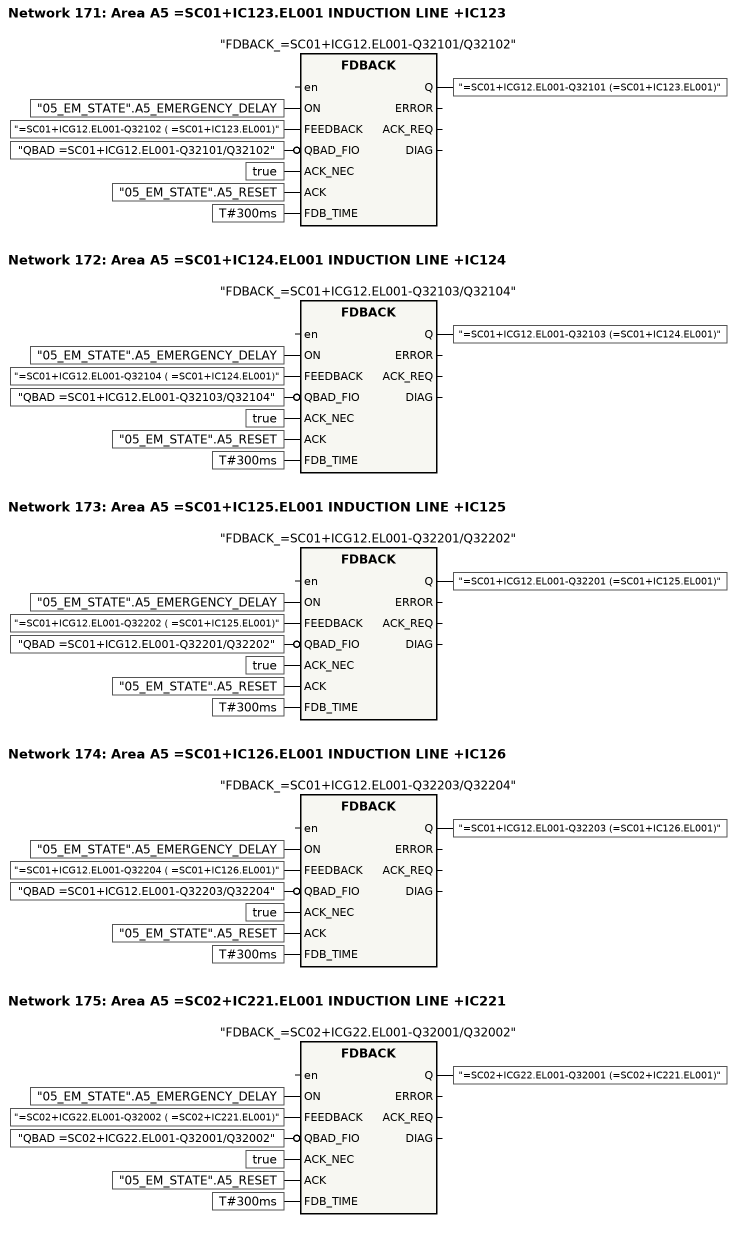
   "FDBACK_=SC01+ICG12.EL001-Q32101/Q32102"(ON := "05_EM_STATE".A5_EMERGENCY_DELAY,   // FDBACK
                           FEEDBACK := "=SC01+ICG12.EL001-Q32102 ( =SC01+IC123.EL001)",
                           QBAD_FIO := NOT "QBAD =SC01+ICG12.EL001-Q32101/Q32102",
                           ACK_NEC := true,
                           ACK := "05_EM_STATE".A5_RESET,
                           FDB_TIME := T#300ms,
                           Q => "=SC01+ICG12.EL001-Q32101 (=SC01+IC123.EL001)");
END_REGION

REGION Network 172: Area A5 =SC01+IC124.EL001 INDUCTION LINE +IC124
   "FDBACK_=SC01+ICG12.EL001-Q32103/Q32104"(ON := "05_EM_STATE".A5_EMERGENCY_DELAY,   // FDBACK
                           FEEDBACK := "=SC01+ICG12.EL001-Q32104 ( =SC01+IC124.EL001)",
                           QBAD_FIO := NOT "QBAD =SC01+ICG12.EL001-Q32103/Q32104",
                           ACK_NEC := true,
                           ACK := "05_EM_STATE".A5_RESET,
                           FDB_TIME := T#300ms,
                           Q => "=SC01+ICG12.EL001-Q32103 (=SC01+IC124.EL001)");
END_REGION

REGION Network 173: Area A5 =SC01+IC125.EL001 INDUCTION LINE +IC125
   "FDBACK_=SC01+ICG12.EL001-Q32201/Q32202"(ON := "05_EM_STATE".A5_EMERGENCY_DELAY,   // FDBACK
                           FEEDBACK := "=SC01+ICG12.EL001-Q32202 ( =SC01+IC125.EL001)",
                           QBAD_FIO := NOT "QBAD =SC01+ICG12.EL001-Q32201/Q32202",
                           ACK_NEC := true,
                           ACK := "05_EM_STATE".A5_RESET,
                           FDB_TIME := T#300ms,
                           Q => "=SC01+ICG12.EL001-Q32201 (=SC01+IC125.EL001)");
END_REGION

REGION Network 174: Area A5 =SC01+IC126.EL001 INDUCTION LINE +IC126
   "FDBACK_=SC01+ICG12.EL001-Q32203/Q32204"(ON := "05_EM_STATE".A5_EMERGENCY_DELAY,   // FDBACK
                           FEEDBACK := "=SC01+ICG12.EL001-Q32204 ( =SC01+IC126.EL001)",
                           QBAD_FIO := NOT "QBAD =SC01+ICG12.EL001-Q32203/Q32204",
                           ACK_NEC := true,
                           ACK := "05_EM_STATE".A5_RESET,
                           FDB_TIME := T#300ms,
                           Q => "=SC01+ICG12.EL001-Q32203 (=SC01+IC126.EL001)");
END_REGION

REGION Network 175: Area A5 =SC02+IC221.EL001 INDUCTION LINE +IC221
   "FDBACK_=SC02+ICG22.EL001-Q32001/Q32002"(ON := "05_EM_STATE".A5_EMERGENCY_DELAY,   // FDBACK
                           FEEDBACK := "=SC02+ICG22.EL001-Q32002 ( =SC02+IC221.EL001)",
                           QBAD_FIO := NOT "QBAD =SC02+ICG22.EL001-Q32001/Q32002",
                           ACK_NEC := true,
                           ACK := "05_EM_STATE".A5_RESET,
                           FDB_TIME := T#300ms,
                           Q => "=SC02+ICG22.EL001-Q32001 (=SC02+IC221.EL001)");
END_REGION

REGION Network 176: Area A5 =SC02+IC222.EL001 INDUCTION LINE +IC222
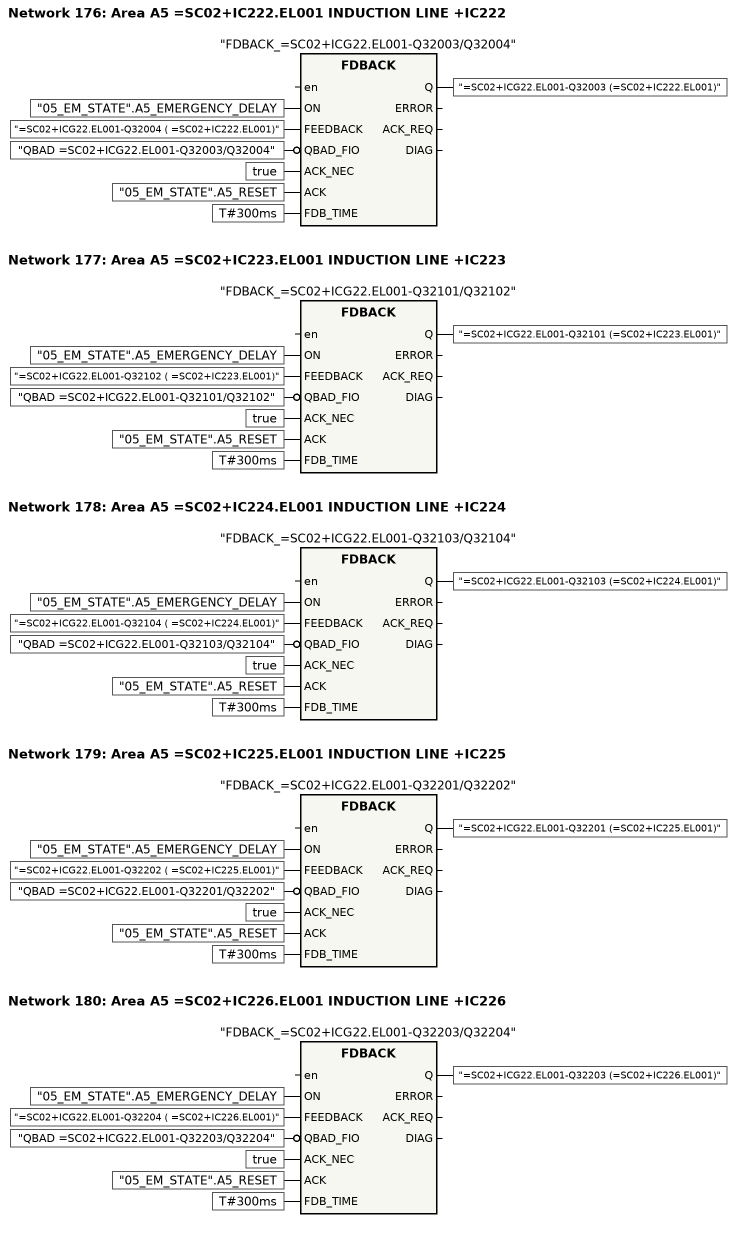
   "FDBACK_=SC02+ICG22.EL001-Q32003/Q32004"(ON := "05_EM_STATE".A5_EMERGENCY_DELAY,   // FDBACK
                           FEEDBACK := "=SC02+ICG22.EL001-Q32004 ( =SC02+IC222.EL001)",
                           QBAD_FIO := NOT "QBAD =SC02+ICG22.EL001-Q32003/Q32004",
                           ACK_NEC := true,
                           ACK := "05_EM_STATE".A5_RESET,
                           FDB_TIME := T#300ms,
                           Q => "=SC02+ICG22.EL001-Q32003 (=SC02+IC222.EL001)");
END_REGION

REGION Network 177: Area A5 =SC02+IC223.EL001 INDUCTION LINE +IC223
   "FDBACK_=SC02+ICG22.EL001-Q32101/Q32102"(ON := "05_EM_STATE".A5_EMERGENCY_DELAY,   // FDBACK
                           FEEDBACK := "=SC02+ICG22.EL001-Q32102 ( =SC02+IC223.EL001)",
                           QBAD_FIO := NOT "QBAD =SC02+ICG22.EL001-Q32101/Q32102",
                           ACK_NEC := true,
                           ACK := "05_EM_STATE".A5_RESET,
                           FDB_TIME := T#300ms,
                           Q => "=SC02+ICG22.EL001-Q32101 (=SC02+IC223.EL001)");
END_REGION

REGION Network 178: Area A5 =SC02+IC224.EL001 INDUCTION LINE +IC224
   "FDBACK_=SC02+ICG22.EL001-Q32103/Q32104"(ON := "05_EM_STATE".A5_EMERGENCY_DELAY,   // FDBACK
                           FEEDBACK := "=SC02+ICG22.EL001-Q32104 ( =SC02+IC224.EL001)",
                           QBAD_FIO := NOT "QBAD =SC02+ICG22.EL001-Q32103/Q32104",
                           ACK_NEC := true,
                           ACK := "05_EM_STATE".A5_RESET,
                           FDB_TIME := T#300ms,
                           Q => "=SC02+ICG22.EL001-Q32103 (=SC02+IC224.EL001)");
END_REGION

REGION Network 179: Area A5 =SC02+IC225.EL001 INDUCTION LINE +IC225
   "FDBACK_=SC02+ICG22.EL001-Q32201/Q32202"(ON := "05_EM_STATE".A5_EMERGENCY_DELAY,   // FDBACK
                           FEEDBACK := "=SC02+ICG22.EL001-Q32202 ( =SC02+IC225.EL001)",
                           QBAD_FIO := NOT "QBAD =SC02+ICG22.EL001-Q32201/Q32202",
                           ACK_NEC := true,
                           ACK := "05_EM_STATE".A5_RESET,
                           FDB_TIME := T#300ms,
                           Q => "=SC02+ICG22.EL001-Q32201 (=SC02+IC225.EL001)");
END_REGION

REGION Network 180: Area A5 =SC02+IC226.EL001 INDUCTION LINE +IC226
   "FDBACK_=SC02+ICG22.EL001-Q32203/Q32204"(ON := "05_EM_STATE".A5_EMERGENCY_DELAY,   // FDBACK
                           FEEDBACK := "=SC02+ICG22.EL001-Q32204 ( =SC02+IC226.EL001)",
                           QBAD_FIO := NOT "QBAD =SC02+ICG22.EL001-Q32203/Q32204",
                           ACK_NEC := true,
                           ACK := "05_EM_STATE".A5_RESET,
                           FDB_TIME := T#300ms,
                           Q => "=SC02+ICG22.EL001-Q32203 (=SC02+IC226.EL001)");
END_REGION

REGION Network 181: Area A5 =SC00+UC213.RB007 - GF003 POWER CUT UC213 LINE
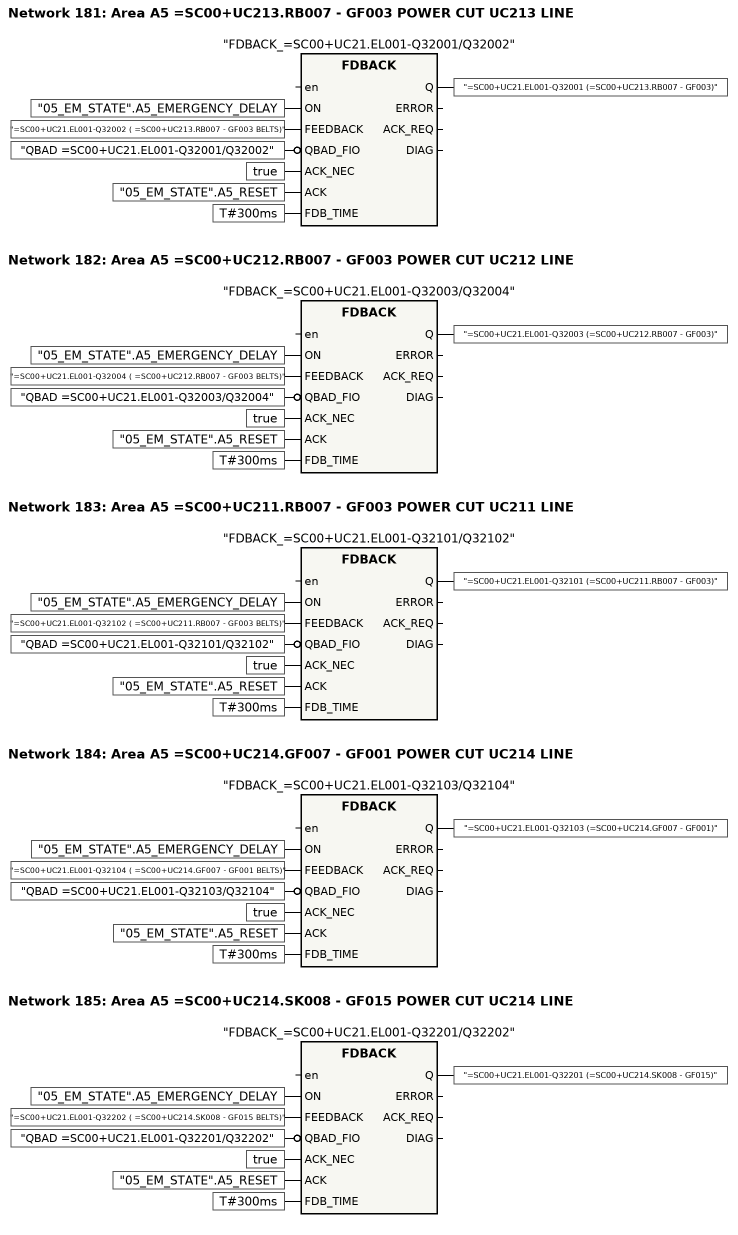
   "FDBACK_=SC00+UC21.EL001-Q32001/Q32002"(ON := "05_EM_STATE".A5_EMERGENCY_DELAY,   // FDBACK
                           FEEDBACK := "=SC00+UC21.EL001-Q32002 ( =SC00+UC213.RB007 - GF003 BELTS)",
                           QBAD_FIO := NOT "QBAD =SC00+UC21.EL001-Q32001/Q32002",
                           ACK_NEC := true,
                           ACK := "05_EM_STATE".A5_RESET,
                           FDB_TIME := T#300ms,
                           Q => "=SC00+UC21.EL001-Q32001 (=SC00+UC213.RB007 - GF003)");
END_REGION

REGION Network 182: Area A5 =SC00+UC212.RB007 - GF003 POWER CUT UC212 LINE
   "FDBACK_=SC00+UC21.EL001-Q32003/Q32004"(ON := "05_EM_STATE".A5_EMERGENCY_DELAY,   // FDBACK
                           FEEDBACK := "=SC00+UC21.EL001-Q32004 ( =SC00+UC212.RB007 - GF003 BELTS)",
                           QBAD_FIO := NOT "QBAD =SC00+UC21.EL001-Q32003/Q32004",
                           ACK_NEC := true,
                           ACK := "05_EM_STATE".A5_RESET,
                           FDB_TIME := T#300ms,
                           Q => "=SC00+UC21.EL001-Q32003 (=SC00+UC212.RB007 - GF003)");
END_REGION

REGION Network 183: Area A5 =SC00+UC211.RB007 - GF003 POWER CUT UC211 LINE
   "FDBACK_=SC00+UC21.EL001-Q32101/Q32102"(ON := "05_EM_STATE".A5_EMERGENCY_DELAY,   // FDBACK
                           FEEDBACK := "=SC00+UC21.EL001-Q32102 ( =SC00+UC211.RB007 - GF003 BELTS)",
                           QBAD_FIO := NOT "QBAD =SC00+UC21.EL001-Q32101/Q32102",
                           ACK_NEC := true,
                           ACK := "05_EM_STATE".A5_RESET,
                           FDB_TIME := T#300ms,
                           Q => "=SC00+UC21.EL001-Q32101 (=SC00+UC211.RB007 - GF003)");
END_REGION

REGION Network 184: Area A5 =SC00+UC214.GF007 - GF001 POWER CUT UC214 LINE
   "FDBACK_=SC00+UC21.EL001-Q32103/Q32104"(ON := "05_EM_STATE".A5_EMERGENCY_DELAY,   // FDBACK
                           FEEDBACK := "=SC00+UC21.EL001-Q32104 ( =SC00+UC214.GF007 - GF001 BELTS)",
                           QBAD_FIO := NOT "QBAD =SC00+UC21.EL001-Q32103/Q32104",
                           ACK_NEC := true,
                           ACK := "05_EM_STATE".A5_RESET,
                           FDB_TIME := T#300ms,
                           Q => "=SC00+UC21.EL001-Q32103 (=SC00+UC214.GF007 - GF001)");
END_REGION

REGION Network 185: Area A5 =SC00+UC214.SK008 - GF015 POWER CUT UC214 LINE
   "FDBACK_=SC00+UC21.EL001-Q32201/Q32202"(ON := "05_EM_STATE".A5_EMERGENCY_DELAY,   // FDBACK
                           FEEDBACK := "=SC00+UC21.EL001-Q32202 ( =SC00+UC214.SK008 - GF015 BELTS)",
                           QBAD_FIO := NOT "QBAD =SC00+UC21.EL001-Q32201/Q32202",
                           ACK_NEC := true,
                           ACK := "05_EM_STATE".A5_RESET,
                           FDB_TIME := T#300ms,
                           Q => "=SC00+UC21.EL001-Q32201 (=SC00+UC214.SK008 - GF015)");
END_REGION

REGION Network 186: Area A5 =SC00+UC214.GF016 - GF018 POWER CUT UC214 LINE
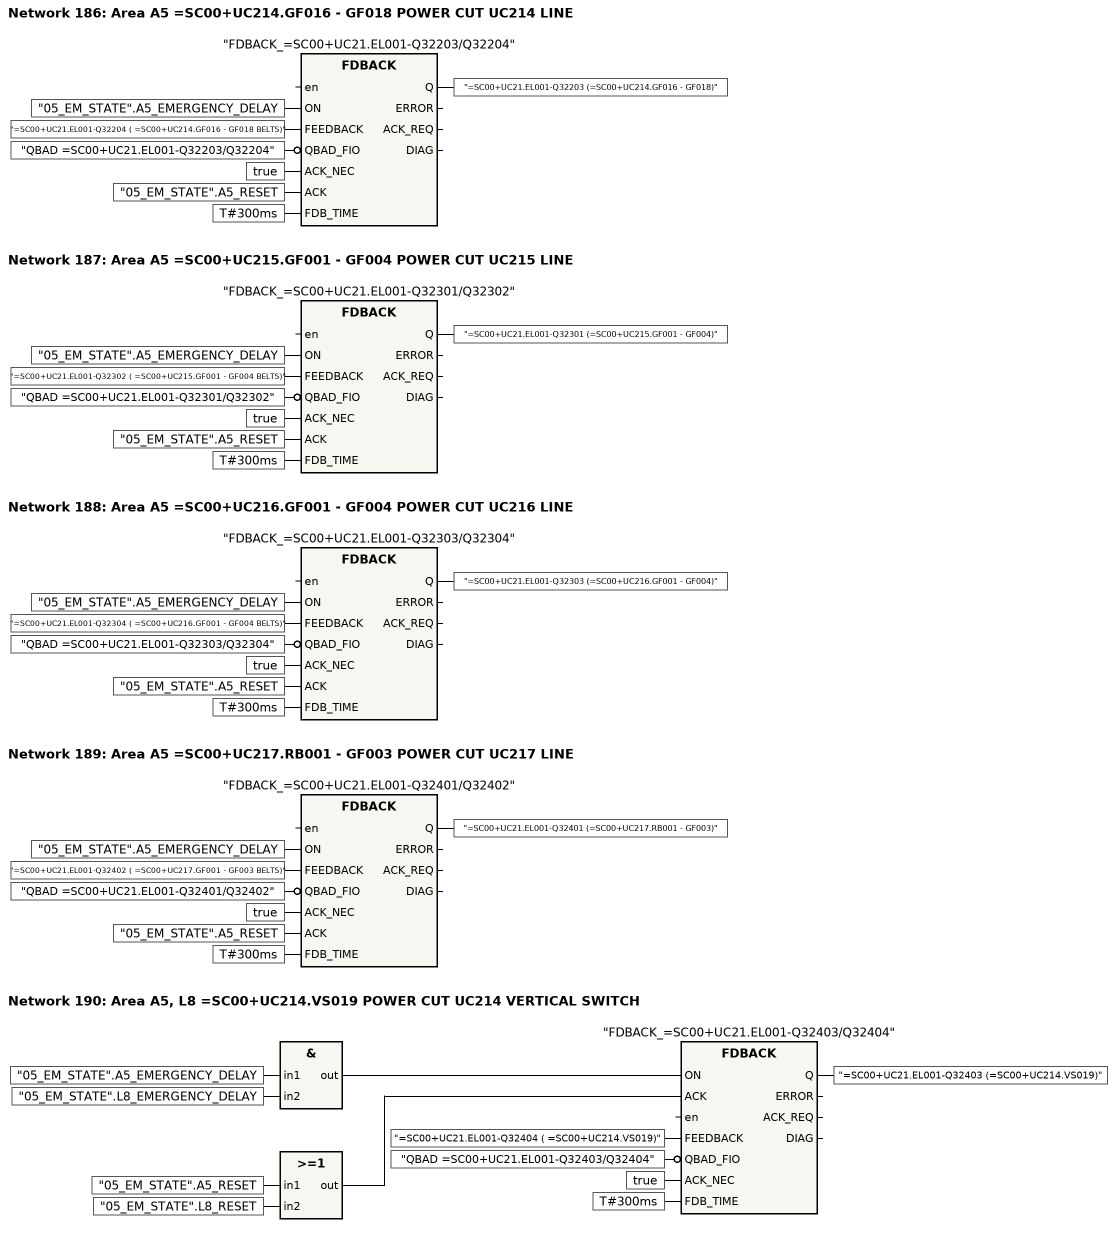
   "FDBACK_=SC00+UC21.EL001-Q32203/Q32204"(ON := "05_EM_STATE".A5_EMERGENCY_DELAY,   // FDBACK
                           FEEDBACK := "=SC00+UC21.EL001-Q32204 ( =SC00+UC214.GF016 - GF018 BELTS)",
                           QBAD_FIO := NOT "QBAD =SC00+UC21.EL001-Q32203/Q32204",
                           ACK_NEC := true,
                           ACK := "05_EM_STATE".A5_RESET,
                           FDB_TIME := T#300ms,
                           Q => "=SC00+UC21.EL001-Q32203 (=SC00+UC214.GF016 - GF018)");
END_REGION

REGION Network 187: Area A5 =SC00+UC215.GF001 - GF004 POWER CUT UC215 LINE
   "FDBACK_=SC00+UC21.EL001-Q32301/Q32302"(ON := "05_EM_STATE".A5_EMERGENCY_DELAY,   // FDBACK
                           FEEDBACK := "=SC00+UC21.EL001-Q32302 ( =SC00+UC215.GF001 - GF004 BELTS)",
                           QBAD_FIO := NOT "QBAD =SC00+UC21.EL001-Q32301/Q32302",
                           ACK_NEC := true,
                           ACK := "05_EM_STATE".A5_RESET,
                           FDB_TIME := T#300ms,
                           Q => "=SC00+UC21.EL001-Q32301 (=SC00+UC215.GF001 - GF004)");
END_REGION

REGION Network 188: Area A5 =SC00+UC216.GF001 - GF004 POWER CUT UC216 LINE
   "FDBACK_=SC00+UC21.EL001-Q32303/Q32304"(ON := "05_EM_STATE".A5_EMERGENCY_DELAY,   // FDBACK
                           FEEDBACK := "=SC00+UC21.EL001-Q32304 ( =SC00+UC216.GF001 - GF004 BELTS)",
                           QBAD_FIO := NOT "QBAD =SC00+UC21.EL001-Q32303/Q32304",
                           ACK_NEC := true,
                           ACK := "05_EM_STATE".A5_RESET,
                           FDB_TIME := T#300ms,
                           Q => "=SC00+UC21.EL001-Q32303 (=SC00+UC216.GF001 - GF004)");
END_REGION

REGION Network 189: Area A5 =SC00+UC217.RB001 - GF003 POWER CUT UC217 LINE
   "FDBACK_=SC00+UC21.EL001-Q32401/Q32402"(ON := "05_EM_STATE".A5_EMERGENCY_DELAY,   // FDBACK
                           FEEDBACK := "=SC00+UC21.EL001-Q32402 ( =SC00+UC217.GF001 - GF003 BELTS)",
                           QBAD_FIO := NOT "QBAD =SC00+UC21.EL001-Q32401/Q32402",
                           ACK_NEC := true,
                           ACK := "05_EM_STATE".A5_RESET,
                           FDB_TIME := T#300ms,
                           Q => "=SC00+UC21.EL001-Q32401 (=SC00+UC217.RB001 - GF003)");
END_REGION

REGION Network 190: Area A5, L8 =SC00+UC214.VS019 POWER CUT UC214 VERTICAL SWITCH
   "FDBACK_=SC00+UC21.EL001-Q32403/Q32404"(ON := "05_EM_STATE".A5_EMERGENCY_DELAY AND "05_EM_STATE".L8_EMERGENCY_DELAY,   // FDBACK
                           ACK := "05_EM_STATE".A5_RESET OR "05_EM_STATE".L8_RESET,
                           FEEDBACK := "=SC00+UC21.EL001-Q32404 ( =SC00+UC214.VS019)",
                           QBAD_FIO := NOT "QBAD =SC00+UC21.EL001-Q32403/Q32404",
                           ACK_NEC := true,
                           FDB_TIME := T#300ms,
                           Q => "=SC00+UC21.EL001-Q32403 (=SC00+UC214.VS019)");
END_REGION

REGION Network 191: Area A5, L8 =SC00+UC214.VS019 VERTICAL SWITCH +UC214
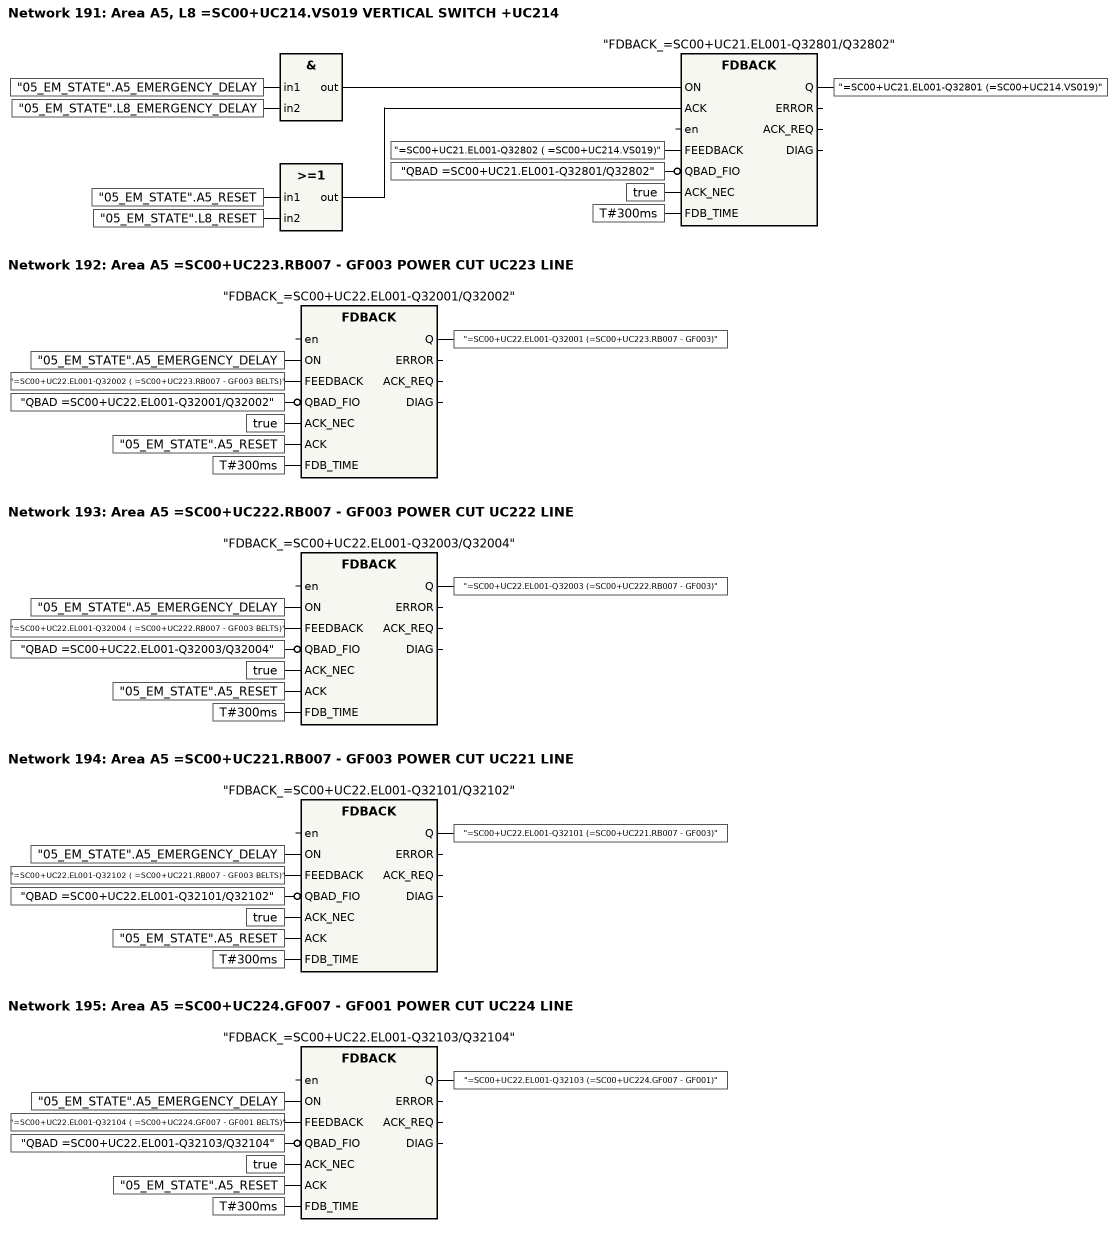
   "FDBACK_=SC00+UC21.EL001-Q32801/Q32802"(ON := "05_EM_STATE".A5_EMERGENCY_DELAY AND "05_EM_STATE".L8_EMERGENCY_DELAY,   // FDBACK
                           ACK := "05_EM_STATE".A5_RESET OR "05_EM_STATE".L8_RESET,
                           FEEDBACK := "=SC00+UC21.EL001-Q32802 ( =SC00+UC214.VS019)",
                           QBAD_FIO := NOT "QBAD =SC00+UC21.EL001-Q32801/Q32802",
                           ACK_NEC := true,
                           FDB_TIME := T#300ms,
                           Q => "=SC00+UC21.EL001-Q32801 (=SC00+UC214.VS019)");
END_REGION

REGION Network 192: Area A5 =SC00+UC223.RB007 - GF003 POWER CUT UC223 LINE
   "FDBACK_=SC00+UC22.EL001-Q32001/Q32002"(ON := "05_EM_STATE".A5_EMERGENCY_DELAY,   // FDBACK
                           FEEDBACK := "=SC00+UC22.EL001-Q32002 ( =SC00+UC223.RB007 - GF003 BELTS)",
                           QBAD_FIO := NOT "QBAD =SC00+UC22.EL001-Q32001/Q32002",
                           ACK_NEC := true,
                           ACK := "05_EM_STATE".A5_RESET,
                           FDB_TIME := T#300ms,
                           Q => "=SC00+UC22.EL001-Q32001 (=SC00+UC223.RB007 - GF003)");
END_REGION

REGION Network 193: Area A5 =SC00+UC222.RB007 - GF003 POWER CUT UC222 LINE
   "FDBACK_=SC00+UC22.EL001-Q32003/Q32004"(ON := "05_EM_STATE".A5_EMERGENCY_DELAY,   // FDBACK
                           FEEDBACK := "=SC00+UC22.EL001-Q32004 ( =SC00+UC222.RB007 - GF003 BELTS)",
                           QBAD_FIO := NOT "QBAD =SC00+UC22.EL001-Q32003/Q32004",
                           ACK_NEC := true,
                           ACK := "05_EM_STATE".A5_RESET,
                           FDB_TIME := T#300ms,
                           Q => "=SC00+UC22.EL001-Q32003 (=SC00+UC222.RB007 - GF003)");
END_REGION

REGION Network 194: Area A5 =SC00+UC221.RB007 - GF003 POWER CUT UC221 LINE
   "FDBACK_=SC00+UC22.EL001-Q32101/Q32102"(ON := "05_EM_STATE".A5_EMERGENCY_DELAY,   // FDBACK
                           FEEDBACK := "=SC00+UC22.EL001-Q32102 ( =SC00+UC221.RB007 - GF003 BELTS)",
                           QBAD_FIO := NOT "QBAD =SC00+UC22.EL001-Q32101/Q32102",
                           ACK_NEC := true,
                           ACK := "05_EM_STATE".A5_RESET,
                           FDB_TIME := T#300ms,
                           Q => "=SC00+UC22.EL001-Q32101 (=SC00+UC221.RB007 - GF003)");
END_REGION

REGION Network 195: Area A5 =SC00+UC224.GF007 - GF001 POWER CUT UC224 LINE
   "FDBACK_=SC00+UC22.EL001-Q32103/Q32104"(ON := "05_EM_STATE".A5_EMERGENCY_DELAY,   // FDBACK
                           FEEDBACK := "=SC00+UC22.EL001-Q32104 ( =SC00+UC224.GF007 - GF001 BELTS)",
                           QBAD_FIO := NOT "QBAD =SC00+UC22.EL001-Q32103/Q32104",
                           ACK_NEC := true,
                           ACK := "05_EM_STATE".A5_RESET,
                           FDB_TIME := T#300ms,
                           Q => "=SC00+UC22.EL001-Q32103 (=SC00+UC224.GF007 - GF001)");
END_REGION

REGION Network 196: Area A5 =SC00+UC224.SK008 - GF015 POWER CUT UC224 LINE
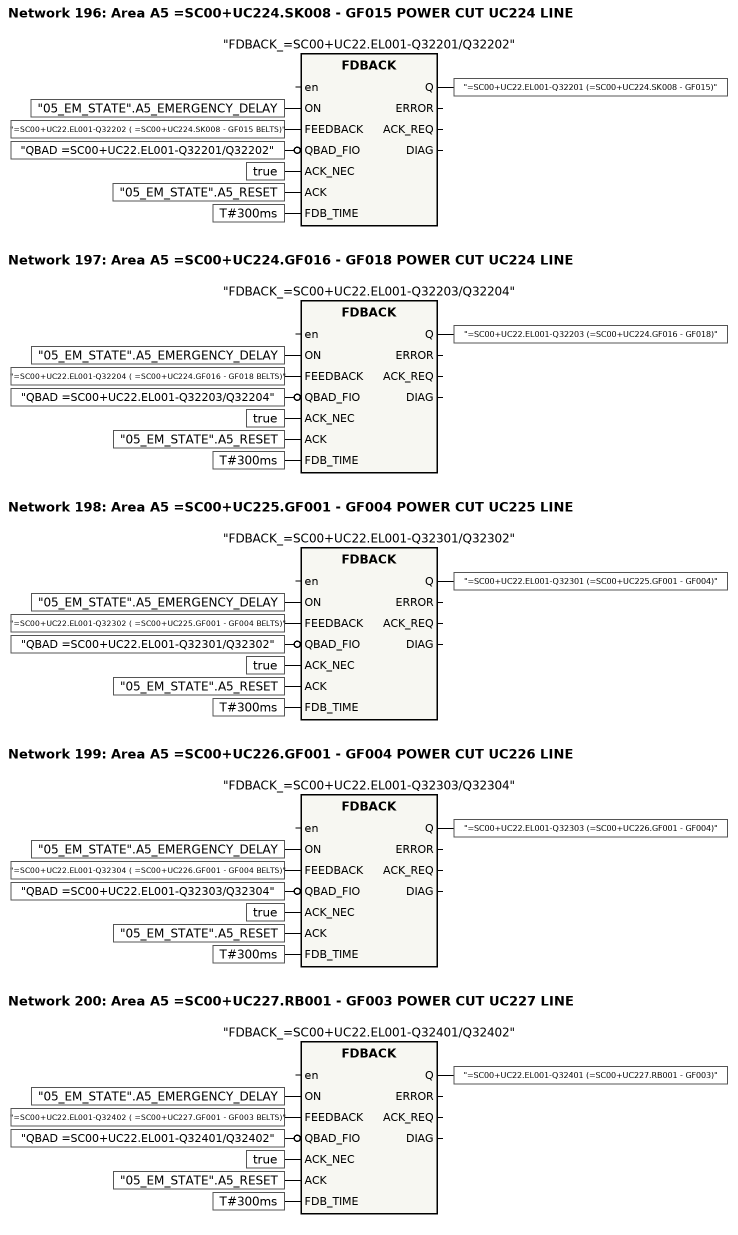
   "FDBACK_=SC00+UC22.EL001-Q32201/Q32202"(ON := "05_EM_STATE".A5_EMERGENCY_DELAY,   // FDBACK
                           FEEDBACK := "=SC00+UC22.EL001-Q32202 ( =SC00+UC224.SK008 - GF015 BELTS)",
                           QBAD_FIO := NOT "QBAD =SC00+UC22.EL001-Q32201/Q32202",
                           ACK_NEC := true,
                           ACK := "05_EM_STATE".A5_RESET,
                           FDB_TIME := T#300ms,
                           Q => "=SC00+UC22.EL001-Q32201 (=SC00+UC224.SK008 - GF015)");
END_REGION

REGION Network 197: Area A5 =SC00+UC224.GF016 - GF018 POWER CUT UC224 LINE
   "FDBACK_=SC00+UC22.EL001-Q32203/Q32204"(ON := "05_EM_STATE".A5_EMERGENCY_DELAY,   // FDBACK
                           FEEDBACK := "=SC00+UC22.EL001-Q32204 ( =SC00+UC224.GF016 - GF018 BELTS)",
                           QBAD_FIO := NOT "QBAD =SC00+UC22.EL001-Q32203/Q32204",
                           ACK_NEC := true,
                           ACK := "05_EM_STATE".A5_RESET,
                           FDB_TIME := T#300ms,
                           Q => "=SC00+UC22.EL001-Q32203 (=SC00+UC224.GF016 - GF018)");
END_REGION

REGION Network 198: Area A5 =SC00+UC225.GF001 - GF004 POWER CUT UC225 LINE
   "FDBACK_=SC00+UC22.EL001-Q32301/Q32302"(ON := "05_EM_STATE".A5_EMERGENCY_DELAY,   // FDBACK
                           FEEDBACK := "=SC00+UC22.EL001-Q32302 ( =SC00+UC225.GF001 - GF004 BELTS)",
                           QBAD_FIO := NOT "QBAD =SC00+UC22.EL001-Q32301/Q32302",
                           ACK_NEC := true,
                           ACK := "05_EM_STATE".A5_RESET,
                           FDB_TIME := T#300ms,
                           Q => "=SC00+UC22.EL001-Q32301 (=SC00+UC225.GF001 - GF004)");
END_REGION

REGION Network 199: Area A5 =SC00+UC226.GF001 - GF004 POWER CUT UC226 LINE
   "FDBACK_=SC00+UC22.EL001-Q32303/Q32304"(ON := "05_EM_STATE".A5_EMERGENCY_DELAY,   // FDBACK
                           FEEDBACK := "=SC00+UC22.EL001-Q32304 ( =SC00+UC226.GF001 - GF004 BELTS)",
                           QBAD_FIO := NOT "QBAD =SC00+UC22.EL001-Q32303/Q32304",
                           ACK_NEC := true,
                           ACK := "05_EM_STATE".A5_RESET,
                           FDB_TIME := T#300ms,
                           Q => "=SC00+UC22.EL001-Q32303 (=SC00+UC226.GF001 - GF004)");
END_REGION

REGION Network 200: Area A5 =SC00+UC227.RB001 - GF003 POWER CUT UC227 LINE
   "FDBACK_=SC00+UC22.EL001-Q32401/Q32402"(ON := "05_EM_STATE".A5_EMERGENCY_DELAY,   // FDBACK
                           FEEDBACK := "=SC00+UC22.EL001-Q32402 ( =SC00+UC227.GF001 - GF003 BELTS)",
                           QBAD_FIO := NOT "QBAD =SC00+UC22.EL001-Q32401/Q32402",
                           ACK_NEC := true,
                           ACK := "05_EM_STATE".A5_RESET,
                           FDB_TIME := T#300ms,
                           Q => "=SC00+UC22.EL001-Q32401 (=SC00+UC227.RB001 - GF003)");
END_REGION

REGION Network 201: Area A5, L9 =SC00+UC224.VS019 POWER CUT UC224 VERTICAL SWITCH
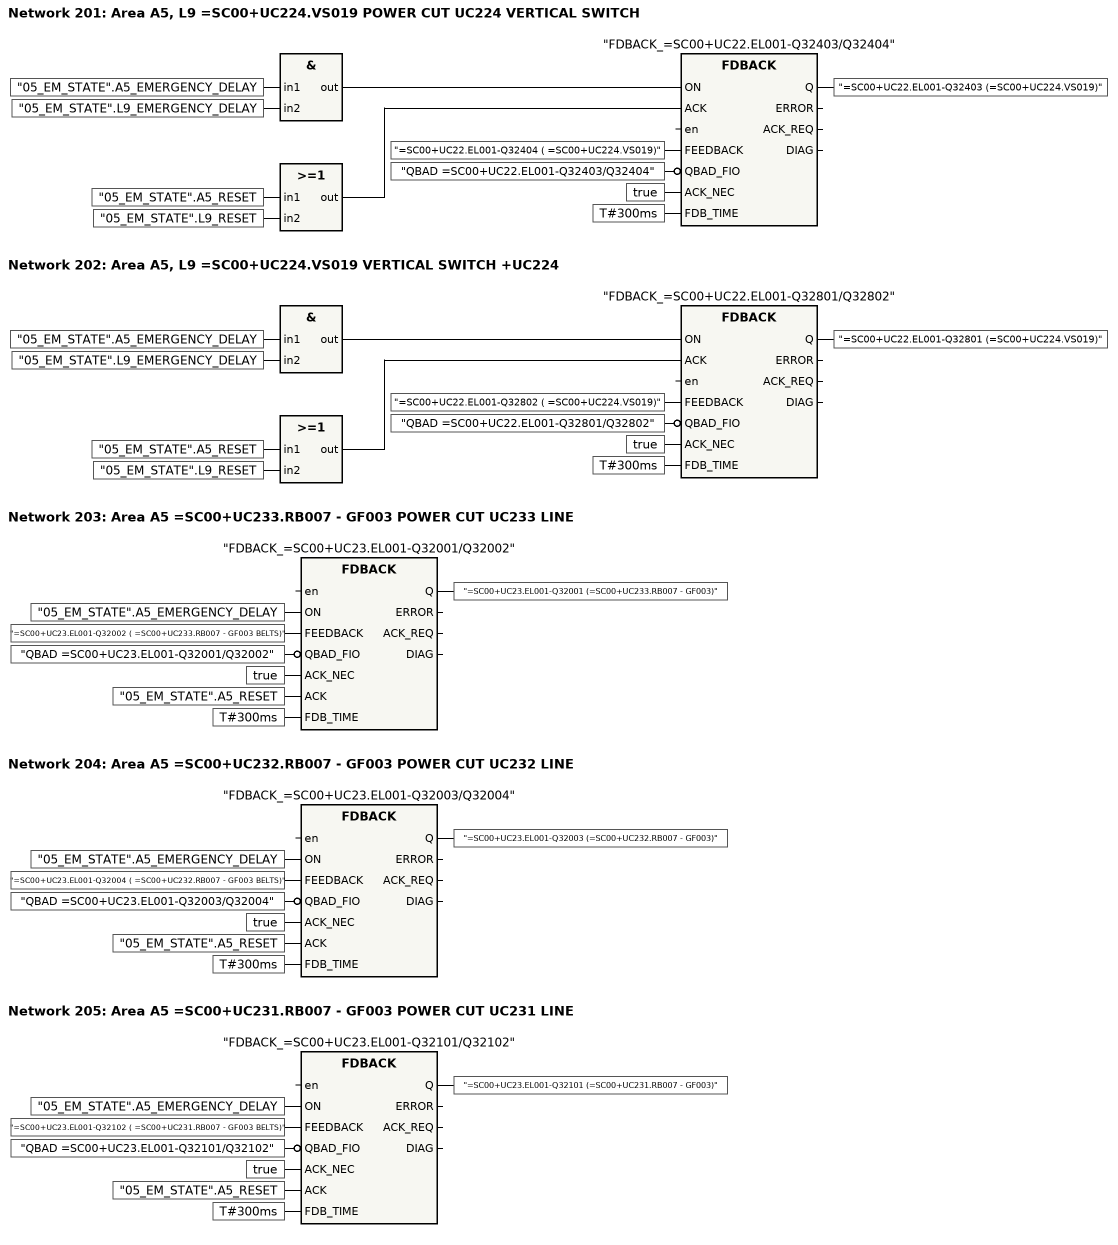
   "FDBACK_=SC00+UC22.EL001-Q32403/Q32404"(ON := "05_EM_STATE".A5_EMERGENCY_DELAY AND "05_EM_STATE".L9_EMERGENCY_DELAY,   // FDBACK
                           ACK := "05_EM_STATE".A5_RESET OR "05_EM_STATE".L9_RESET,
                           FEEDBACK := "=SC00+UC22.EL001-Q32404 ( =SC00+UC224.VS019)",
                           QBAD_FIO := NOT "QBAD =SC00+UC22.EL001-Q32403/Q32404",
                           ACK_NEC := true,
                           FDB_TIME := T#300ms,
                           Q => "=SC00+UC22.EL001-Q32403 (=SC00+UC224.VS019)");
END_REGION

REGION Network 202: Area A5, L9 =SC00+UC224.VS019 VERTICAL SWITCH +UC224
   "FDBACK_=SC00+UC22.EL001-Q32801/Q32802"(ON := "05_EM_STATE".A5_EMERGENCY_DELAY AND "05_EM_STATE".L9_EMERGENCY_DELAY,   // FDBACK
                           ACK := "05_EM_STATE".A5_RESET OR "05_EM_STATE".L9_RESET,
                           FEEDBACK := "=SC00+UC22.EL001-Q32802 ( =SC00+UC224.VS019)",
                           QBAD_FIO := NOT "QBAD =SC00+UC22.EL001-Q32801/Q32802",
                           ACK_NEC := true,
                           FDB_TIME := T#300ms,
                           Q => "=SC00+UC22.EL001-Q32801 (=SC00+UC224.VS019)");
END_REGION

REGION Network 203: Area A5 =SC00+UC233.RB007 - GF003 POWER CUT UC233 LINE
   "FDBACK_=SC00+UC23.EL001-Q32001/Q32002"(ON := "05_EM_STATE".A5_EMERGENCY_DELAY,   // FDBACK
                           FEEDBACK := "=SC00+UC23.EL001-Q32002 ( =SC00+UC233.RB007 - GF003 BELTS)",
                           QBAD_FIO := NOT "QBAD =SC00+UC23.EL001-Q32001/Q32002",
                           ACK_NEC := true,
                           ACK := "05_EM_STATE".A5_RESET,
                           FDB_TIME := T#300ms,
                           Q => "=SC00+UC23.EL001-Q32001 (=SC00+UC233.RB007 - GF003)");
END_REGION

REGION Network 204: Area A5 =SC00+UC232.RB007 - GF003 POWER CUT UC232 LINE
   "FDBACK_=SC00+UC23.EL001-Q32003/Q32004"(ON := "05_EM_STATE".A5_EMERGENCY_DELAY,   // FDBACK
                           FEEDBACK := "=SC00+UC23.EL001-Q32004 ( =SC00+UC232.RB007 - GF003 BELTS)",
                           QBAD_FIO := NOT "QBAD =SC00+UC23.EL001-Q32003/Q32004",
                           ACK_NEC := true,
                           ACK := "05_EM_STATE".A5_RESET,
                           FDB_TIME := T#300ms,
                           Q => "=SC00+UC23.EL001-Q32003 (=SC00+UC232.RB007 - GF003)");
END_REGION

REGION Network 205: Area A5 =SC00+UC231.RB007 - GF003 POWER CUT UC231 LINE
   "FDBACK_=SC00+UC23.EL001-Q32101/Q32102"(ON := "05_EM_STATE".A5_EMERGENCY_DELAY,   // FDBACK
                           FEEDBACK := "=SC00+UC23.EL001-Q32102 ( =SC00+UC231.RB007 - GF003 BELTS)",
                           QBAD_FIO := NOT "QBAD =SC00+UC23.EL001-Q32101/Q32102",
                           ACK_NEC := true,
                           ACK := "05_EM_STATE".A5_RESET,
                           FDB_TIME := T#300ms,
                           Q => "=SC00+UC23.EL001-Q32101 (=SC00+UC231.RB007 - GF003)");
END_REGION

REGION Network 206: Area A5 =SC00+UC234.GF007 - GF001 POWER CUT UC234 LINE
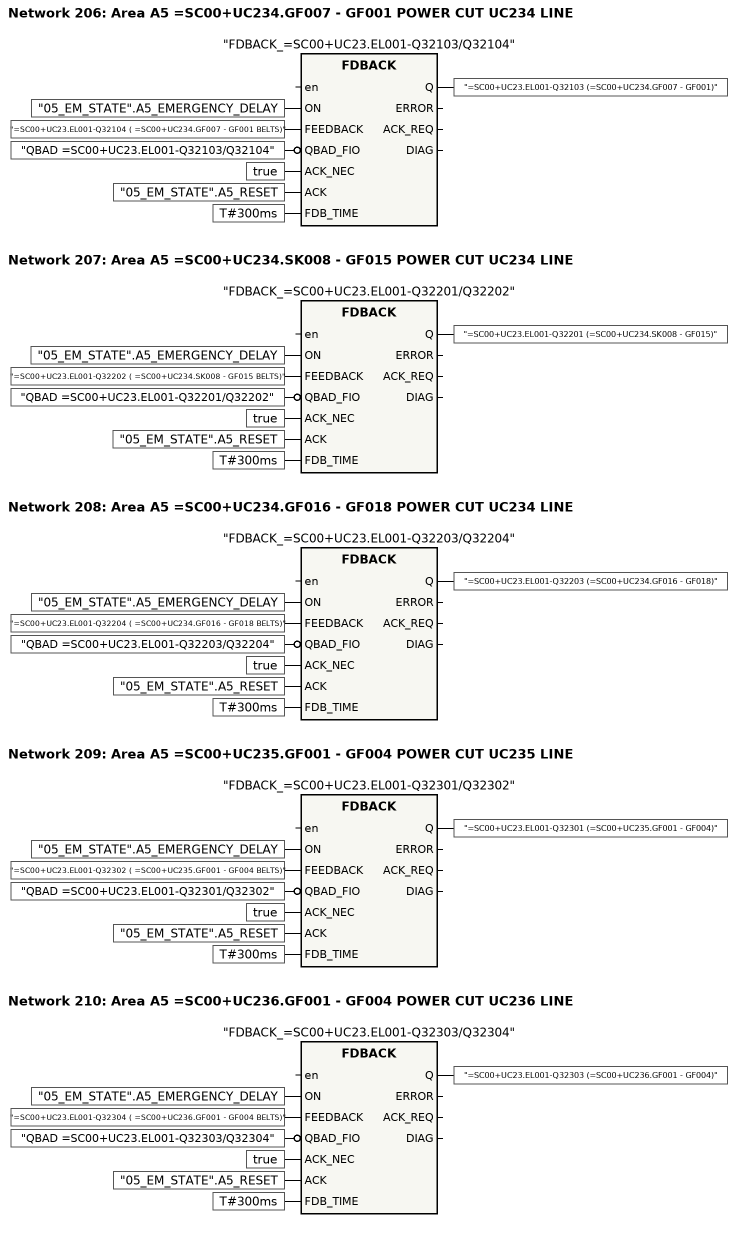
   "FDBACK_=SC00+UC23.EL001-Q32103/Q32104"(ON := "05_EM_STATE".A5_EMERGENCY_DELAY,   // FDBACK
                           FEEDBACK := "=SC00+UC23.EL001-Q32104 ( =SC00+UC234.GF007 - GF001 BELTS)",
                           QBAD_FIO := NOT "QBAD =SC00+UC23.EL001-Q32103/Q32104",
                           ACK_NEC := true,
                           ACK := "05_EM_STATE".A5_RESET,
                           FDB_TIME := T#300ms,
                           Q => "=SC00+UC23.EL001-Q32103 (=SC00+UC234.GF007 - GF001)");
END_REGION

REGION Network 207: Area A5 =SC00+UC234.SK008 - GF015 POWER CUT UC234 LINE
   "FDBACK_=SC00+UC23.EL001-Q32201/Q32202"(ON := "05_EM_STATE".A5_EMERGENCY_DELAY,   // FDBACK
                           FEEDBACK := "=SC00+UC23.EL001-Q32202 ( =SC00+UC234.SK008 - GF015 BELTS)",
                           QBAD_FIO := NOT "QBAD =SC00+UC23.EL001-Q32201/Q32202",
                           ACK_NEC := true,
                           ACK := "05_EM_STATE".A5_RESET,
                           FDB_TIME := T#300ms,
                           Q => "=SC00+UC23.EL001-Q32201 (=SC00+UC234.SK008 - GF015)");
END_REGION

REGION Network 208: Area A5 =SC00+UC234.GF016 - GF018 POWER CUT UC234 LINE
   "FDBACK_=SC00+UC23.EL001-Q32203/Q32204"(ON := "05_EM_STATE".A5_EMERGENCY_DELAY,   // FDBACK
                           FEEDBACK := "=SC00+UC23.EL001-Q32204 ( =SC00+UC234.GF016 - GF018 BELTS)",
                           QBAD_FIO := NOT "QBAD =SC00+UC23.EL001-Q32203/Q32204",
                           ACK_NEC := true,
                           ACK := "05_EM_STATE".A5_RESET,
                           FDB_TIME := T#300ms,
                           Q => "=SC00+UC23.EL001-Q32203 (=SC00+UC234.GF016 - GF018)");
END_REGION

REGION Network 209: Area A5 =SC00+UC235.GF001 - GF004 POWER CUT UC235 LINE
   "FDBACK_=SC00+UC23.EL001-Q32301/Q32302"(ON := "05_EM_STATE".A5_EMERGENCY_DELAY,   // FDBACK
                           FEEDBACK := "=SC00+UC23.EL001-Q32302 ( =SC00+UC235.GF001 - GF004 BELTS)",
                           QBAD_FIO := NOT "QBAD =SC00+UC23.EL001-Q32301/Q32302",
                           ACK_NEC := true,
                           ACK := "05_EM_STATE".A5_RESET,
                           FDB_TIME := T#300ms,
                           Q => "=SC00+UC23.EL001-Q32301 (=SC00+UC235.GF001 - GF004)");
END_REGION

REGION Network 210: Area A5 =SC00+UC236.GF001 - GF004 POWER CUT UC236 LINE
   "FDBACK_=SC00+UC23.EL001-Q32303/Q32304"(ON := "05_EM_STATE".A5_EMERGENCY_DELAY,   // FDBACK
                           FEEDBACK := "=SC00+UC23.EL001-Q32304 ( =SC00+UC236.GF001 - GF004 BELTS)",
                           QBAD_FIO := NOT "QBAD =SC00+UC23.EL001-Q32303/Q32304",
                           ACK_NEC := true,
                           ACK := "05_EM_STATE".A5_RESET,
                           FDB_TIME := T#300ms,
                           Q => "=SC00+UC23.EL001-Q32303 (=SC00+UC236.GF001 - GF004)");
END_REGION

REGION Network 211: Area A5 =SC00+UC237.RB001 - GF003 POWER CUT UC237 LINE
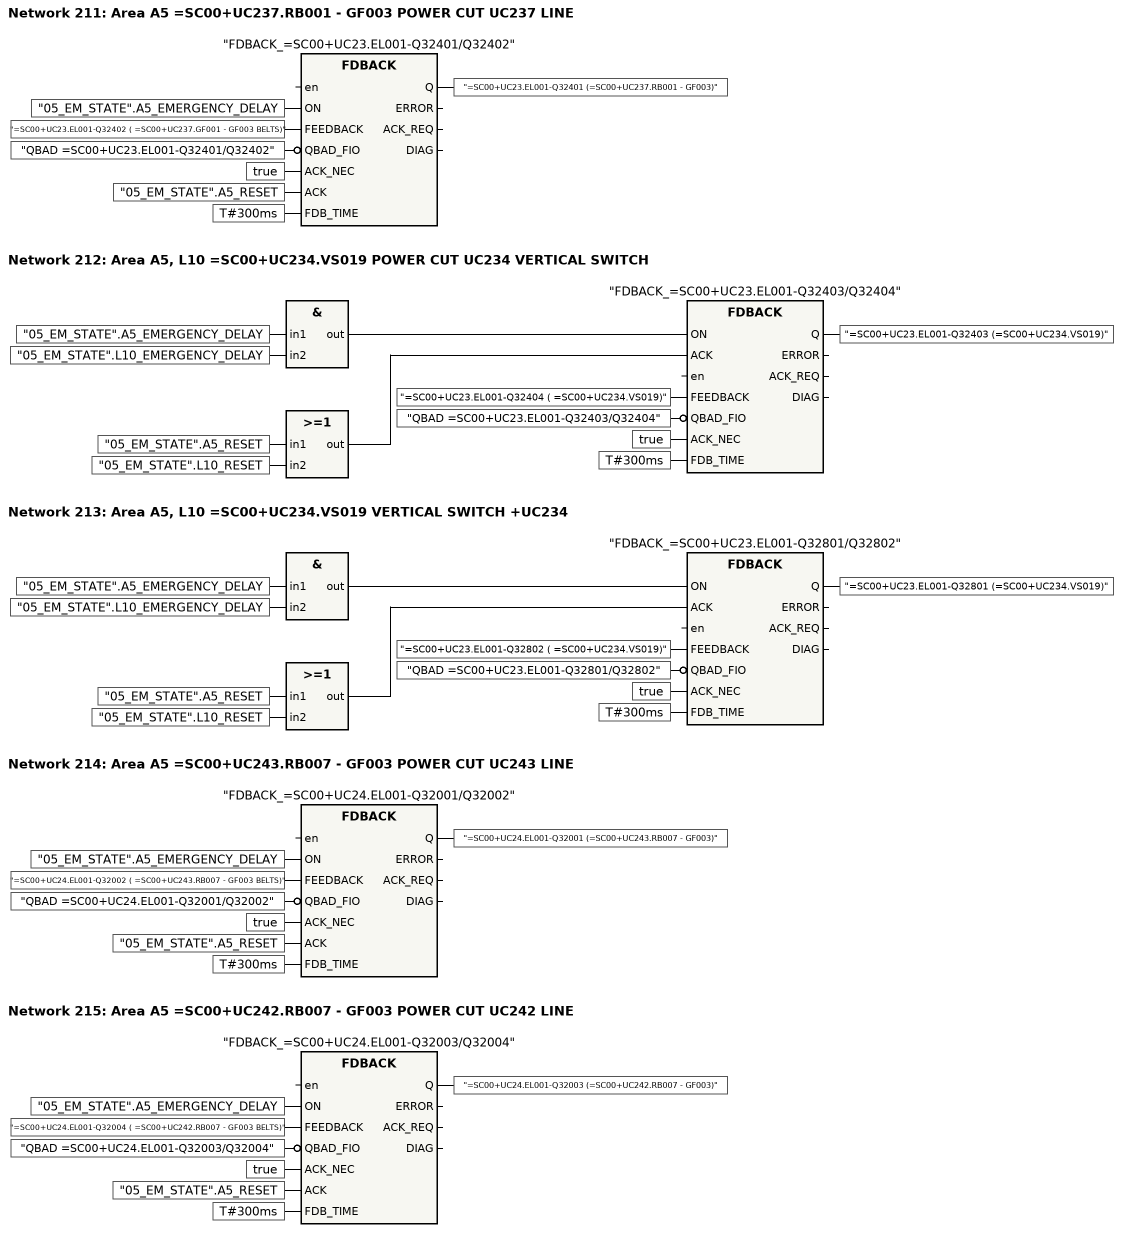
   "FDBACK_=SC00+UC23.EL001-Q32401/Q32402"(ON := "05_EM_STATE".A5_EMERGENCY_DELAY,   // FDBACK
                           FEEDBACK := "=SC00+UC23.EL001-Q32402 ( =SC00+UC237.GF001 - GF003 BELTS)",
                           QBAD_FIO := NOT "QBAD =SC00+UC23.EL001-Q32401/Q32402",
                           ACK_NEC := true,
                           ACK := "05_EM_STATE".A5_RESET,
                           FDB_TIME := T#300ms,
                           Q => "=SC00+UC23.EL001-Q32401 (=SC00+UC237.RB001 - GF003)");
END_REGION

REGION Network 212: Area A5, L10 =SC00+UC234.VS019 POWER CUT UC234 VERTICAL SWITCH
   "FDBACK_=SC00+UC23.EL001-Q32403/Q32404"(ON := "05_EM_STATE".A5_EMERGENCY_DELAY AND "05_EM_STATE".L10_EMERGENCY_DELAY,   // FDBACK
                           ACK := "05_EM_STATE".A5_RESET OR "05_EM_STATE".L10_RESET,
                           FEEDBACK := "=SC00+UC23.EL001-Q32404 ( =SC00+UC234.VS019)",
                           QBAD_FIO := NOT "QBAD =SC00+UC23.EL001-Q32403/Q32404",
                           ACK_NEC := true,
                           FDB_TIME := T#300ms,
                           Q => "=SC00+UC23.EL001-Q32403 (=SC00+UC234.VS019)");
END_REGION

REGION Network 213: Area A5, L10 =SC00+UC234.VS019 VERTICAL SWITCH +UC234
   "FDBACK_=SC00+UC23.EL001-Q32801/Q32802"(ON := "05_EM_STATE".A5_EMERGENCY_DELAY AND "05_EM_STATE".L10_EMERGENCY_DELAY,   // FDBACK
                           ACK := "05_EM_STATE".A5_RESET OR "05_EM_STATE".L10_RESET,
                           FEEDBACK := "=SC00+UC23.EL001-Q32802 ( =SC00+UC234.VS019)",
                           QBAD_FIO := NOT "QBAD =SC00+UC23.EL001-Q32801/Q32802",
                           ACK_NEC := true,
                           FDB_TIME := T#300ms,
                           Q => "=SC00+UC23.EL001-Q32801 (=SC00+UC234.VS019)");
END_REGION

REGION Network 214: Area A5 =SC00+UC243.RB007 - GF003 POWER CUT UC243 LINE
   "FDBACK_=SC00+UC24.EL001-Q32001/Q32002"(ON := "05_EM_STATE".A5_EMERGENCY_DELAY,   // FDBACK
                           FEEDBACK := "=SC00+UC24.EL001-Q32002 ( =SC00+UC243.RB007 - GF003 BELTS)",
                           QBAD_FIO := NOT "QBAD =SC00+UC24.EL001-Q32001/Q32002",
                           ACK_NEC := true,
                           ACK := "05_EM_STATE".A5_RESET,
                           FDB_TIME := T#300ms,
                           Q => "=SC00+UC24.EL001-Q32001 (=SC00+UC243.RB007 - GF003)");
END_REGION

REGION Network 215: Area A5 =SC00+UC242.RB007 - GF003 POWER CUT UC242 LINE
   "FDBACK_=SC00+UC24.EL001-Q32003/Q32004"(ON := "05_EM_STATE".A5_EMERGENCY_DELAY,   // FDBACK
                           FEEDBACK := "=SC00+UC24.EL001-Q32004 ( =SC00+UC242.RB007 - GF003 BELTS)",
                           QBAD_FIO := NOT "QBAD =SC00+UC24.EL001-Q32003/Q32004",
                           ACK_NEC := true,
                           ACK := "05_EM_STATE".A5_RESET,
                           FDB_TIME := T#300ms,
                           Q => "=SC00+UC24.EL001-Q32003 (=SC00+UC242.RB007 - GF003)");
END_REGION

REGION Network 216: Area A5 =SC00+UC241.RB007 - GF003 POWER CUT UC241 LINE
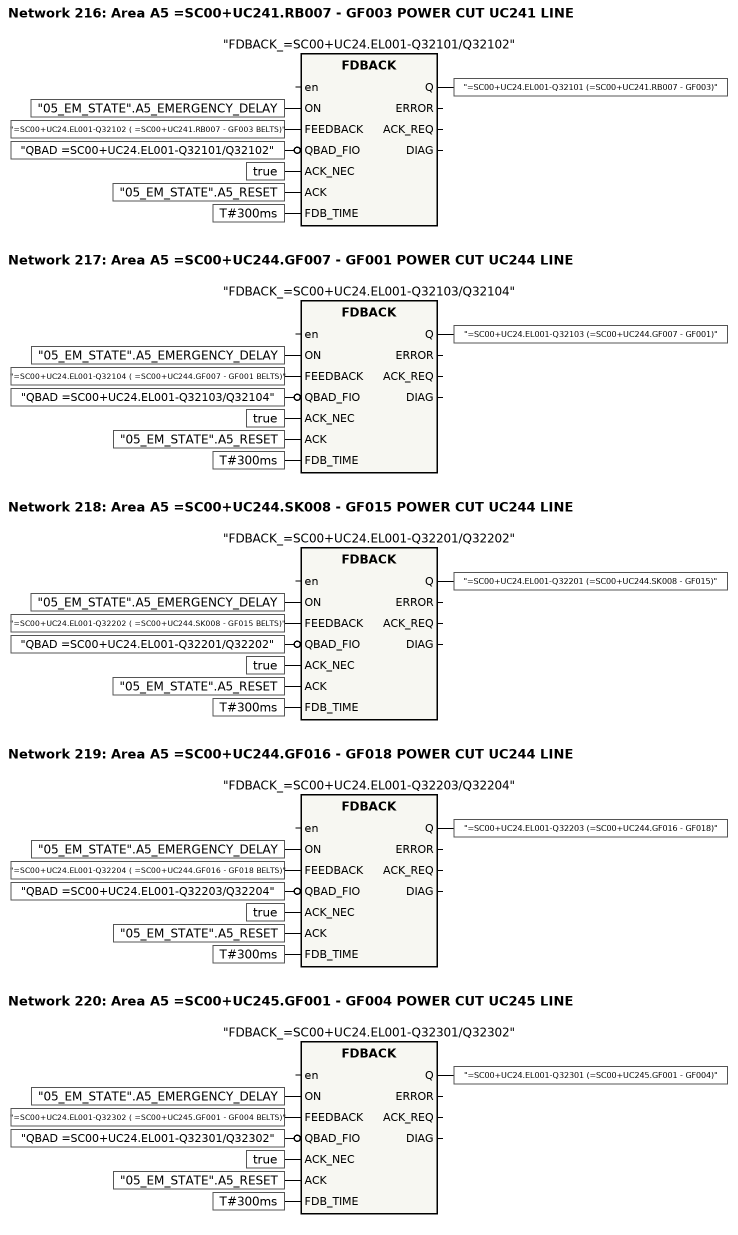
   "FDBACK_=SC00+UC24.EL001-Q32101/Q32102"(ON := "05_EM_STATE".A5_EMERGENCY_DELAY,   // FDBACK
                           FEEDBACK := "=SC00+UC24.EL001-Q32102 ( =SC00+UC241.RB007 - GF003 BELTS)",
                           QBAD_FIO := NOT "QBAD =SC00+UC24.EL001-Q32101/Q32102",
                           ACK_NEC := true,
                           ACK := "05_EM_STATE".A5_RESET,
                           FDB_TIME := T#300ms,
                           Q => "=SC00+UC24.EL001-Q32101 (=SC00+UC241.RB007 - GF003)");
END_REGION

REGION Network 217: Area A5 =SC00+UC244.GF007 - GF001 POWER CUT UC244 LINE
   "FDBACK_=SC00+UC24.EL001-Q32103/Q32104"(ON := "05_EM_STATE".A5_EMERGENCY_DELAY,   // FDBACK
                           FEEDBACK := "=SC00+UC24.EL001-Q32104 ( =SC00+UC244.GF007 - GF001 BELTS)",
                           QBAD_FIO := NOT "QBAD =SC00+UC24.EL001-Q32103/Q32104",
                           ACK_NEC := true,
                           ACK := "05_EM_STATE".A5_RESET,
                           FDB_TIME := T#300ms,
                           Q => "=SC00+UC24.EL001-Q32103 (=SC00+UC244.GF007 - GF001)");
END_REGION

REGION Network 218: Area A5 =SC00+UC244.SK008 - GF015 POWER CUT UC244 LINE
   "FDBACK_=SC00+UC24.EL001-Q32201/Q32202"(ON := "05_EM_STATE".A5_EMERGENCY_DELAY,   // FDBACK
                           FEEDBACK := "=SC00+UC24.EL001-Q32202 ( =SC00+UC244.SK008 - GF015 BELTS)",
                           QBAD_FIO := NOT "QBAD =SC00+UC24.EL001-Q32201/Q32202",
                           ACK_NEC := true,
                           ACK := "05_EM_STATE".A5_RESET,
                           FDB_TIME := T#300ms,
                           Q => "=SC00+UC24.EL001-Q32201 (=SC00+UC244.SK008 - GF015)");
END_REGION

REGION Network 219: Area A5 =SC00+UC244.GF016 - GF018 POWER CUT UC244 LINE
   "FDBACK_=SC00+UC24.EL001-Q32203/Q32204"(ON := "05_EM_STATE".A5_EMERGENCY_DELAY,   // FDBACK
                           FEEDBACK := "=SC00+UC24.EL001-Q32204 ( =SC00+UC244.GF016 - GF018 BELTS)",
                           QBAD_FIO := NOT "QBAD =SC00+UC24.EL001-Q32203/Q32204",
                           ACK_NEC := true,
                           ACK := "05_EM_STATE".A5_RESET,
                           FDB_TIME := T#300ms,
                           Q => "=SC00+UC24.EL001-Q32203 (=SC00+UC244.GF016 - GF018)");
END_REGION

REGION Network 220: Area A5 =SC00+UC245.GF001 - GF004 POWER CUT UC245 LINE
   "FDBACK_=SC00+UC24.EL001-Q32301/Q32302"(ON := "05_EM_STATE".A5_EMERGENCY_DELAY,   // FDBACK
                           FEEDBACK := "=SC00+UC24.EL001-Q32302 ( =SC00+UC245.GF001 - GF004 BELTS)",
                           QBAD_FIO := NOT "QBAD =SC00+UC24.EL001-Q32301/Q32302",
                           ACK_NEC := true,
                           ACK := "05_EM_STATE".A5_RESET,
                           FDB_TIME := T#300ms,
                           Q => "=SC00+UC24.EL001-Q32301 (=SC00+UC245.GF001 - GF004)");
END_REGION

REGION Network 221: Area A5 =SC00+UC246.GF001 - GF004 POWER CUT UC246 LINE
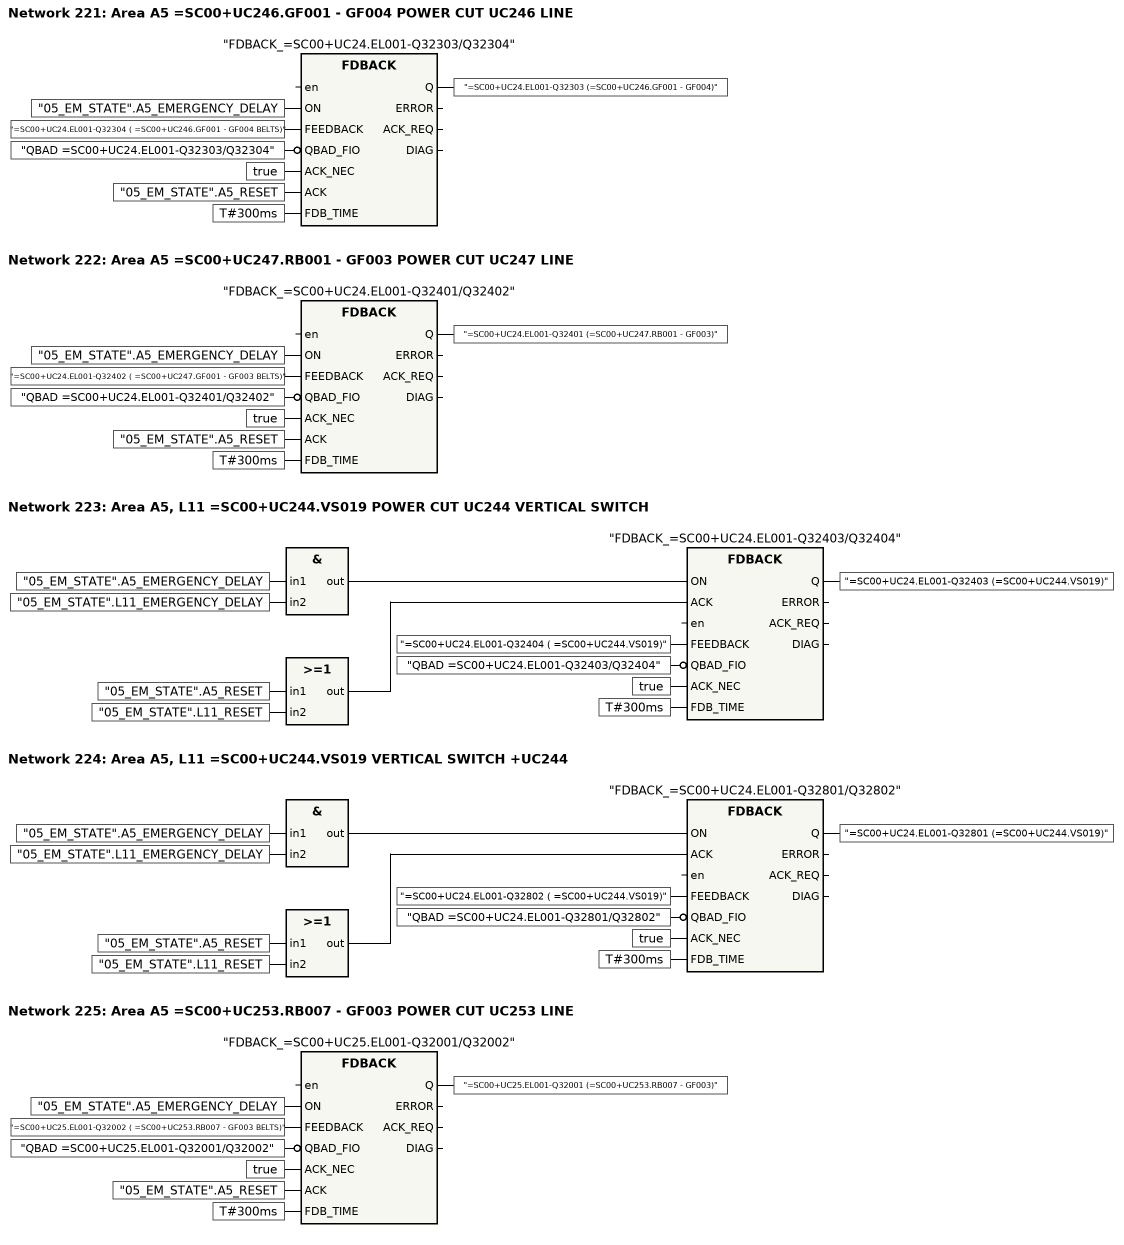
   "FDBACK_=SC00+UC24.EL001-Q32303/Q32304"(ON := "05_EM_STATE".A5_EMERGENCY_DELAY,   // FDBACK
                           FEEDBACK := "=SC00+UC24.EL001-Q32304 ( =SC00+UC246.GF001 - GF004 BELTS)",
                           QBAD_FIO := NOT "QBAD =SC00+UC24.EL001-Q32303/Q32304",
                           ACK_NEC := true,
                           ACK := "05_EM_STATE".A5_RESET,
                           FDB_TIME := T#300ms,
                           Q => "=SC00+UC24.EL001-Q32303 (=SC00+UC246.GF001 - GF004)");
END_REGION

REGION Network 222: Area A5 =SC00+UC247.RB001 - GF003 POWER CUT UC247 LINE
   "FDBACK_=SC00+UC24.EL001-Q32401/Q32402"(ON := "05_EM_STATE".A5_EMERGENCY_DELAY,   // FDBACK
                           FEEDBACK := "=SC00+UC24.EL001-Q32402 ( =SC00+UC247.GF001 - GF003 BELTS)",
                           QBAD_FIO := NOT "QBAD =SC00+UC24.EL001-Q32401/Q32402",
                           ACK_NEC := true,
                           ACK := "05_EM_STATE".A5_RESET,
                           FDB_TIME := T#300ms,
                           Q => "=SC00+UC24.EL001-Q32401 (=SC00+UC247.RB001 - GF003)");
END_REGION

REGION Network 223: Area A5, L11 =SC00+UC244.VS019 POWER CUT UC244 VERTICAL SWITCH
   "FDBACK_=SC00+UC24.EL001-Q32403/Q32404"(ON := "05_EM_STATE".A5_EMERGENCY_DELAY AND "05_EM_STATE".L11_EMERGENCY_DELAY,   // FDBACK
                           ACK := "05_EM_STATE".A5_RESET OR "05_EM_STATE".L11_RESET,
                           FEEDBACK := "=SC00+UC24.EL001-Q32404 ( =SC00+UC244.VS019)",
                           QBAD_FIO := NOT "QBAD =SC00+UC24.EL001-Q32403/Q32404",
                           ACK_NEC := true,
                           FDB_TIME := T#300ms,
                           Q => "=SC00+UC24.EL001-Q32403 (=SC00+UC244.VS019)");
END_REGION

REGION Network 224: Area A5, L11 =SC00+UC244.VS019 VERTICAL SWITCH +UC244
   "FDBACK_=SC00+UC24.EL001-Q32801/Q32802"(ON := "05_EM_STATE".A5_EMERGENCY_DELAY AND "05_EM_STATE".L11_EMERGENCY_DELAY,   // FDBACK
                           ACK := "05_EM_STATE".A5_RESET OR "05_EM_STATE".L11_RESET,
                           FEEDBACK := "=SC00+UC24.EL001-Q32802 ( =SC00+UC244.VS019)",
                           QBAD_FIO := NOT "QBAD =SC00+UC24.EL001-Q32801/Q32802",
                           ACK_NEC := true,
                           FDB_TIME := T#300ms,
                           Q => "=SC00+UC24.EL001-Q32801 (=SC00+UC244.VS019)");
END_REGION

REGION Network 225: Area A5 =SC00+UC253.RB007 - GF003 POWER CUT UC253 LINE
   "FDBACK_=SC00+UC25.EL001-Q32001/Q32002"(ON := "05_EM_STATE".A5_EMERGENCY_DELAY,   // FDBACK
                           FEEDBACK := "=SC00+UC25.EL001-Q32002 ( =SC00+UC253.RB007 - GF003 BELTS)",
                           QBAD_FIO := NOT "QBAD =SC00+UC25.EL001-Q32001/Q32002",
                           ACK_NEC := true,
                           ACK := "05_EM_STATE".A5_RESET,
                           FDB_TIME := T#300ms,
                           Q => "=SC00+UC25.EL001-Q32001 (=SC00+UC253.RB007 - GF003)");
END_REGION

REGION Network 226: Area A5 =SC00+UC252.RB007 - GF003 POWER CUT UC252 LINE
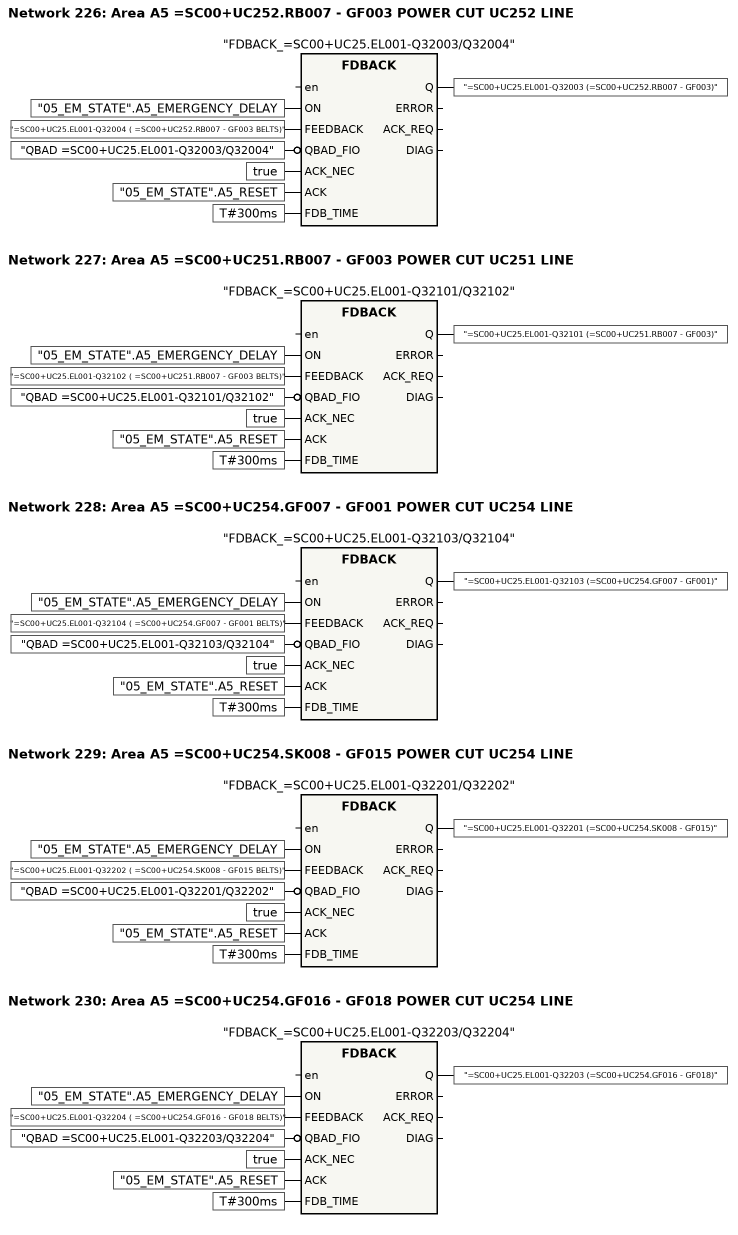
   "FDBACK_=SC00+UC25.EL001-Q32003/Q32004"(ON := "05_EM_STATE".A5_EMERGENCY_DELAY,   // FDBACK
                           FEEDBACK := "=SC00+UC25.EL001-Q32004 ( =SC00+UC252.RB007 - GF003 BELTS)",
                           QBAD_FIO := NOT "QBAD =SC00+UC25.EL001-Q32003/Q32004",
                           ACK_NEC := true,
                           ACK := "05_EM_STATE".A5_RESET,
                           FDB_TIME := T#300ms,
                           Q => "=SC00+UC25.EL001-Q32003 (=SC00+UC252.RB007 - GF003)");
END_REGION

REGION Network 227: Area A5 =SC00+UC251.RB007 - GF003 POWER CUT UC251 LINE
   "FDBACK_=SC00+UC25.EL001-Q32101/Q32102"(ON := "05_EM_STATE".A5_EMERGENCY_DELAY,   // FDBACK
                           FEEDBACK := "=SC00+UC25.EL001-Q32102 ( =SC00+UC251.RB007 - GF003 BELTS)",
                           QBAD_FIO := NOT "QBAD =SC00+UC25.EL001-Q32101/Q32102",
                           ACK_NEC := true,
                           ACK := "05_EM_STATE".A5_RESET,
                           FDB_TIME := T#300ms,
                           Q => "=SC00+UC25.EL001-Q32101 (=SC00+UC251.RB007 - GF003)");
END_REGION

REGION Network 228: Area A5 =SC00+UC254.GF007 - GF001 POWER CUT UC254 LINE
   "FDBACK_=SC00+UC25.EL001-Q32103/Q32104"(ON := "05_EM_STATE".A5_EMERGENCY_DELAY,   // FDBACK
                           FEEDBACK := "=SC00+UC25.EL001-Q32104 ( =SC00+UC254.GF007 - GF001 BELTS)",
                           QBAD_FIO := NOT "QBAD =SC00+UC25.EL001-Q32103/Q32104",
                           ACK_NEC := true,
                           ACK := "05_EM_STATE".A5_RESET,
                           FDB_TIME := T#300ms,
                           Q => "=SC00+UC25.EL001-Q32103 (=SC00+UC254.GF007 - GF001)");
END_REGION

REGION Network 229: Area A5 =SC00+UC254.SK008 - GF015 POWER CUT UC254 LINE
   "FDBACK_=SC00+UC25.EL001-Q32201/Q32202"(ON := "05_EM_STATE".A5_EMERGENCY_DELAY,   // FDBACK
                           FEEDBACK := "=SC00+UC25.EL001-Q32202 ( =SC00+UC254.SK008 - GF015 BELTS)",
                           QBAD_FIO := NOT "QBAD =SC00+UC25.EL001-Q32201/Q32202",
                           ACK_NEC := true,
                           ACK := "05_EM_STATE".A5_RESET,
                           FDB_TIME := T#300ms,
                           Q => "=SC00+UC25.EL001-Q32201 (=SC00+UC254.SK008 - GF015)");
END_REGION

REGION Network 230: Area A5 =SC00+UC254.GF016 - GF018 POWER CUT UC254 LINE
   "FDBACK_=SC00+UC25.EL001-Q32203/Q32204"(ON := "05_EM_STATE".A5_EMERGENCY_DELAY,   // FDBACK
                           FEEDBACK := "=SC00+UC25.EL001-Q32204 ( =SC00+UC254.GF016 - GF018 BELTS)",
                           QBAD_FIO := NOT "QBAD =SC00+UC25.EL001-Q32203/Q32204",
                           ACK_NEC := true,
                           ACK := "05_EM_STATE".A5_RESET,
                           FDB_TIME := T#300ms,
                           Q => "=SC00+UC25.EL001-Q32203 (=SC00+UC254.GF016 - GF018)");
END_REGION

REGION Network 231: Area A5 =SC00+UC255.GF001 - GF004 POWER CUT UC255 LINE
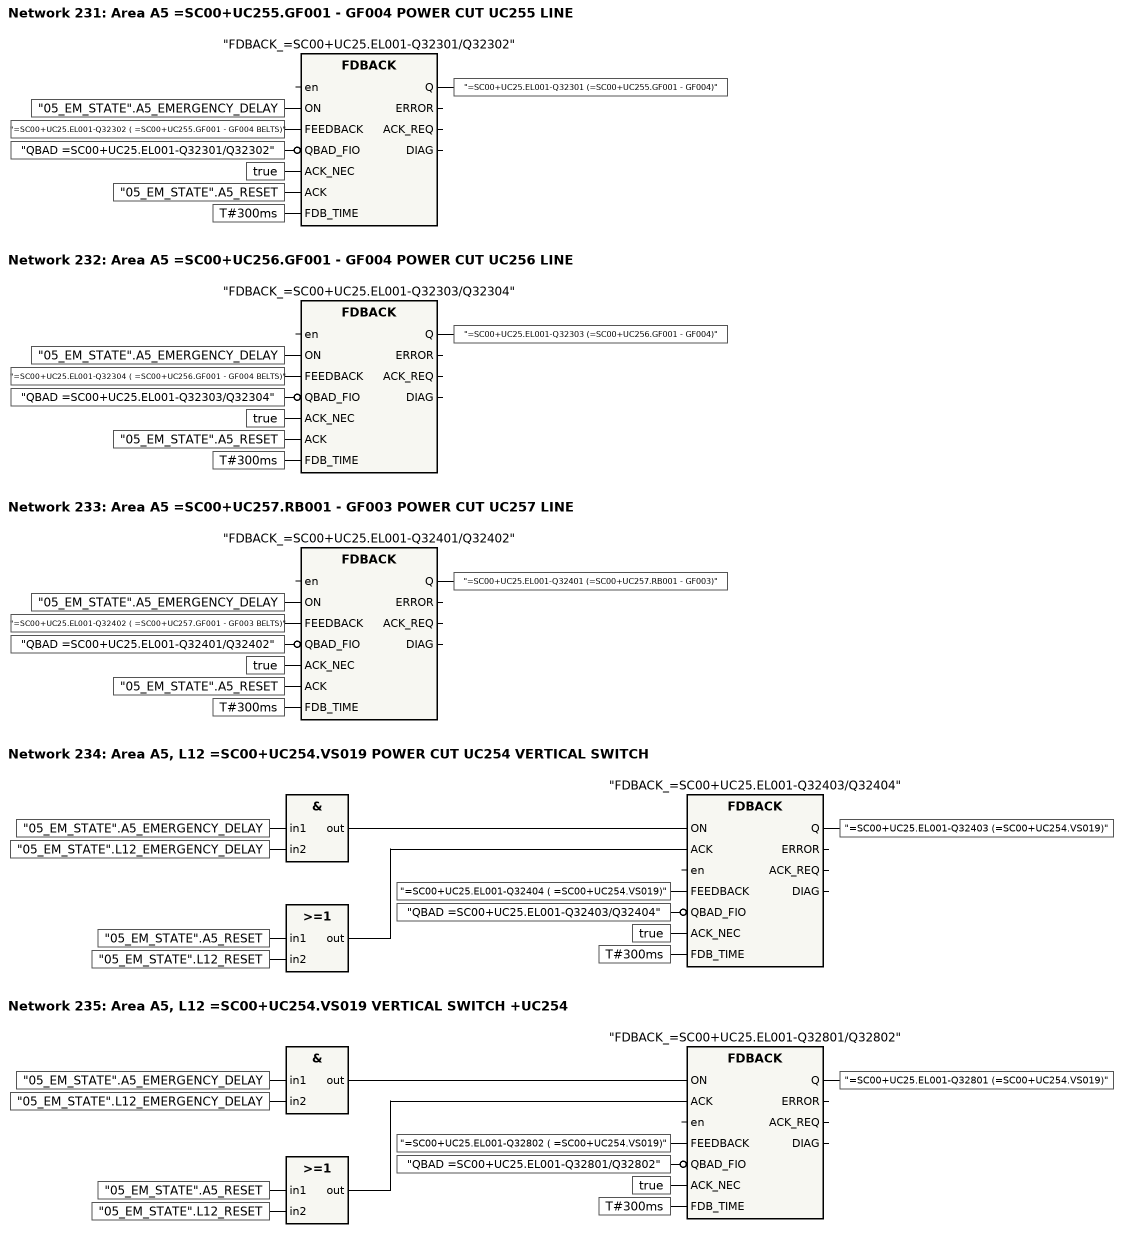
   "FDBACK_=SC00+UC25.EL001-Q32301/Q32302"(ON := "05_EM_STATE".A5_EMERGENCY_DELAY,   // FDBACK
                           FEEDBACK := "=SC00+UC25.EL001-Q32302 ( =SC00+UC255.GF001 - GF004 BELTS)",
                           QBAD_FIO := NOT "QBAD =SC00+UC25.EL001-Q32301/Q32302",
                           ACK_NEC := true,
                           ACK := "05_EM_STATE".A5_RESET,
                           FDB_TIME := T#300ms,
                           Q => "=SC00+UC25.EL001-Q32301 (=SC00+UC255.GF001 - GF004)");
END_REGION

REGION Network 232: Area A5 =SC00+UC256.GF001 - GF004 POWER CUT UC256 LINE
   "FDBACK_=SC00+UC25.EL001-Q32303/Q32304"(ON := "05_EM_STATE".A5_EMERGENCY_DELAY,   // FDBACK
                           FEEDBACK := "=SC00+UC25.EL001-Q32304 ( =SC00+UC256.GF001 - GF004 BELTS)",
                           QBAD_FIO := NOT "QBAD =SC00+UC25.EL001-Q32303/Q32304",
                           ACK_NEC := true,
                           ACK := "05_EM_STATE".A5_RESET,
                           FDB_TIME := T#300ms,
                           Q => "=SC00+UC25.EL001-Q32303 (=SC00+UC256.GF001 - GF004)");
END_REGION

REGION Network 233: Area A5 =SC00+UC257.RB001 - GF003 POWER CUT UC257 LINE
   "FDBACK_=SC00+UC25.EL001-Q32401/Q32402"(ON := "05_EM_STATE".A5_EMERGENCY_DELAY,   // FDBACK
                           FEEDBACK := "=SC00+UC25.EL001-Q32402 ( =SC00+UC257.GF001 - GF003 BELTS)",
                           QBAD_FIO := NOT "QBAD =SC00+UC25.EL001-Q32401/Q32402",
                           ACK_NEC := true,
                           ACK := "05_EM_STATE".A5_RESET,
                           FDB_TIME := T#300ms,
                           Q => "=SC00+UC25.EL001-Q32401 (=SC00+UC257.RB001 - GF003)");
END_REGION

REGION Network 234: Area A5, L12 =SC00+UC254.VS019 POWER CUT UC254 VERTICAL SWITCH
   "FDBACK_=SC00+UC25.EL001-Q32403/Q32404"(ON := "05_EM_STATE".A5_EMERGENCY_DELAY AND "05_EM_STATE".L12_EMERGENCY_DELAY,   // FDBACK
                           ACK := "05_EM_STATE".A5_RESET OR "05_EM_STATE".L12_RESET,
                           FEEDBACK := "=SC00+UC25.EL001-Q32404 ( =SC00+UC254.VS019)",
                           QBAD_FIO := NOT "QBAD =SC00+UC25.EL001-Q32403/Q32404",
                           ACK_NEC := true,
                           FDB_TIME := T#300ms,
                           Q => "=SC00+UC25.EL001-Q32403 (=SC00+UC254.VS019)");
END_REGION

REGION Network 235: Area A5, L12 =SC00+UC254.VS019 VERTICAL SWITCH +UC254
   "FDBACK_=SC00+UC25.EL001-Q32801/Q32802"(ON := "05_EM_STATE".A5_EMERGENCY_DELAY AND "05_EM_STATE".L12_EMERGENCY_DELAY,   // FDBACK
                           ACK := "05_EM_STATE".A5_RESET OR "05_EM_STATE".L12_RESET,
                           FEEDBACK := "=SC00+UC25.EL001-Q32802 ( =SC00+UC254.VS019)",
                           QBAD_FIO := NOT "QBAD =SC00+UC25.EL001-Q32801/Q32802",
                           ACK_NEC := true,
                           FDB_TIME := T#300ms,
                           Q => "=SC00+UC25.EL001-Q32801 (=SC00+UC254.VS019)");
END_REGION

REGION Network 236: Area A5 =SC00+UC263.RB007 - GF003 POWER CUT UC263 LINE
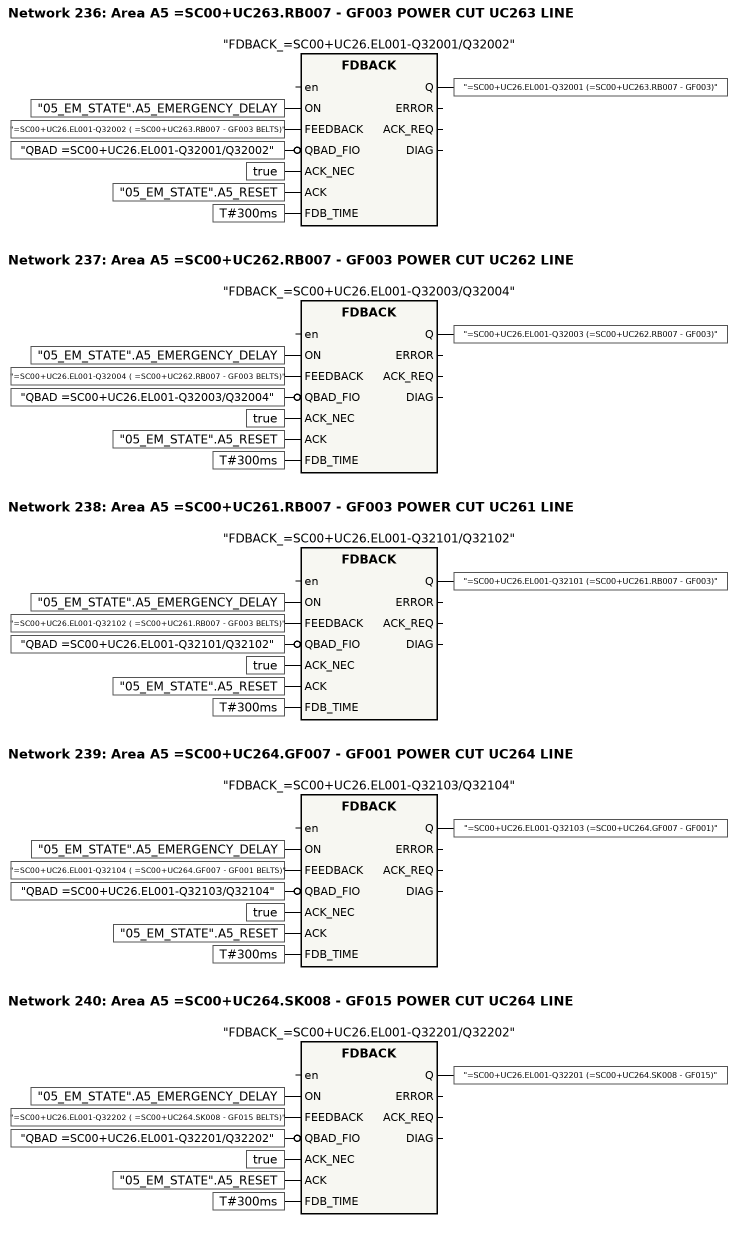
   "FDBACK_=SC00+UC26.EL001-Q32001/Q32002"(ON := "05_EM_STATE".A5_EMERGENCY_DELAY,   // FDBACK
                           FEEDBACK := "=SC00+UC26.EL001-Q32002 ( =SC00+UC263.RB007 - GF003 BELTS)",
                           QBAD_FIO := NOT "QBAD =SC00+UC26.EL001-Q32001/Q32002",
                           ACK_NEC := true,
                           ACK := "05_EM_STATE".A5_RESET,
                           FDB_TIME := T#300ms,
                           Q => "=SC00+UC26.EL001-Q32001 (=SC00+UC263.RB007 - GF003)");
END_REGION

REGION Network 237: Area A5 =SC00+UC262.RB007 - GF003 POWER CUT UC262 LINE
   "FDBACK_=SC00+UC26.EL001-Q32003/Q32004"(ON := "05_EM_STATE".A5_EMERGENCY_DELAY,   // FDBACK
                           FEEDBACK := "=SC00+UC26.EL001-Q32004 ( =SC00+UC262.RB007 - GF003 BELTS)",
                           QBAD_FIO := NOT "QBAD =SC00+UC26.EL001-Q32003/Q32004",
                           ACK_NEC := true,
                           ACK := "05_EM_STATE".A5_RESET,
                           FDB_TIME := T#300ms,
                           Q => "=SC00+UC26.EL001-Q32003 (=SC00+UC262.RB007 - GF003)");
END_REGION

REGION Network 238: Area A5 =SC00+UC261.RB007 - GF003 POWER CUT UC261 LINE
   "FDBACK_=SC00+UC26.EL001-Q32101/Q32102"(ON := "05_EM_STATE".A5_EMERGENCY_DELAY,   // FDBACK
                           FEEDBACK := "=SC00+UC26.EL001-Q32102 ( =SC00+UC261.RB007 - GF003 BELTS)",
                           QBAD_FIO := NOT "QBAD =SC00+UC26.EL001-Q32101/Q32102",
                           ACK_NEC := true,
                           ACK := "05_EM_STATE".A5_RESET,
                           FDB_TIME := T#300ms,
                           Q => "=SC00+UC26.EL001-Q32101 (=SC00+UC261.RB007 - GF003)");
END_REGION

REGION Network 239: Area A5 =SC00+UC264.GF007 - GF001 POWER CUT UC264 LINE
   "FDBACK_=SC00+UC26.EL001-Q32103/Q32104"(ON := "05_EM_STATE".A5_EMERGENCY_DELAY,   // FDBACK
                           FEEDBACK := "=SC00+UC26.EL001-Q32104 ( =SC00+UC264.GF007 - GF001 BELTS)",
                           QBAD_FIO := NOT "QBAD =SC00+UC26.EL001-Q32103/Q32104",
                           ACK_NEC := true,
                           ACK := "05_EM_STATE".A5_RESET,
                           FDB_TIME := T#300ms,
                           Q => "=SC00+UC26.EL001-Q32103 (=SC00+UC264.GF007 - GF001)");
END_REGION

REGION Network 240: Area A5 =SC00+UC264.SK008 - GF015 POWER CUT UC264 LINE
   "FDBACK_=SC00+UC26.EL001-Q32201/Q32202"(ON := "05_EM_STATE".A5_EMERGENCY_DELAY,   // FDBACK
                           FEEDBACK := "=SC00+UC26.EL001-Q32202 ( =SC00+UC264.SK008 - GF015 BELTS)",
                           QBAD_FIO := NOT "QBAD =SC00+UC26.EL001-Q32201/Q32202",
                           ACK_NEC := true,
                           ACK := "05_EM_STATE".A5_RESET,
                           FDB_TIME := T#300ms,
                           Q => "=SC00+UC26.EL001-Q32201 (=SC00+UC264.SK008 - GF015)");
END_REGION

REGION Network 241: Area A5 =SC00+UC264.GF016 - GF018 POWER CUT UC264 LINE
